//     PlcTask Inputs/GVL_iXlinker.EtherCAT_Master_BKCUCX.TcTerminals210_EK1100_1.TcTerminals210_1BK1250.A_0132_KL_1032_2_Ch_Input_48V_3_0ms.Channel_1.Input <-> Channel 1/Input
//     PlcTask Inputs/GVL_iXlinker.EtherCAT_Master_BKCUCX.TcTerminals210_EK1100_1.TcTerminals210_1BK1250.A_0132_KL_1032_2_Ch_Input_48V_3_0ms.Channel_2.Input <-> Channel 2/Input
//   PLC/PLC Instance <-> EtherCAT Master BKCUCX/TcTerminals210_EK1100_1/TcTerminals210_1BK1250/A_0133(KL 1052, 2 Ch. Input +/- (24V, 3.0ms))
//     PlcTask Inputs/GVL_iXlinker.EtherCAT_Master_BKCUCX.TcTerminals210_EK1100_1.TcTerminals210_1BK1250.A_0133_KL_1052_2_Ch_Input_24V_3_0ms.Channel_1.Input <-> Channel 1/Input
//     PlcTask Inputs/GVL_iXlinker.EtherCAT_Master_BKCUCX.TcTerminals210_EK1100_1.TcTerminals210_1BK1250.A_0133_KL_1052_2_Ch_Input_24V_3_0ms.Channel_2.Input <-> Channel 2/Input
//   PLC/PLC Instance <-> EtherCAT Master BKCUCX/TcTerminals210_EK1100_1/TcTerminals210_1BK1250/A_0134(KL 1104, 4 Ch. Input (24V, 3.0ms))
//     PlcTask Inputs/GVL_iXlinker.EtherCAT_Master_BKCUCX.TcTerminals210_EK1100_1.TcTerminals210_1BK1250.A_0134_KL_1104_4_Ch_Input_24V_3_0ms.Channel_1.Input <-> Channel 1/Input
//     PlcTask Inputs/GVL_iXlinker.EtherCAT_Master_BKCUCX.TcTerminals210_EK1100_1.TcTerminals210_1BK1250.A_0134_KL_1104_4_Ch_Input_24V_3_0ms.Channel_2.Input <-> Channel 2/Input
//     PlcTask Inputs/GVL_iXlinker.EtherCAT_Master_BKCUCX.TcTerminals210_EK1100_1.TcTerminals210_1BK1250.A_0134_KL_1104_4_Ch_Input_24V_3_0ms.Channel_3.Input <-> Channel 3/Input
//     PlcTask Inputs/GVL_iXlinker.EtherCAT_Master_BKCUCX.TcTerminals210_EK1100_1.TcTerminals210_1BK1250.A_0134_KL_1104_4_Ch_Input_24V_3_0ms.Channel_4.Input <-> Channel 4/Input
//   PLC/PLC Instance <-> EtherCAT Master BKCUCX/TcTerminals210_EK1100_1/TcTerminals210_1BK1250/A_0135(KL 1114, 4 Ch. Input (24V, 0.2ms))
//     PlcTask Inputs/GVL_iXlinker.EtherCAT_Master_BKCUCX.TcTerminals210_EK1100_1.TcTerminals210_1BK1250.A_0135_KL_1114_4_Ch_Input_24V_0_2ms.Channel_1.Input <-> Channel 1/Input
//     PlcTask Inputs/GVL_iXlinker.EtherCAT_Master_BKCUCX.TcTerminals210_EK1100_1.TcTerminals210_1BK1250.A_0135_KL_1114_4_Ch_Input_24V_0_2ms.Channel_2.Input <-> Channel 2/Input
//     PlcTask Inputs/GVL_iXlinker.EtherCAT_Master_BKCUCX.TcTerminals210_EK1100_1.TcTerminals210_1BK1250.A_0135_KL_1114_4_Ch_Input_24V_0_2ms.Channel_3.Input <-> Channel 3/Input
//     PlcTask Inputs/GVL_iXlinker.EtherCAT_Master_BKCUCX.TcTerminals210_EK1100_1.TcTerminals210_1BK1250.A_0135_KL_1114_4_Ch_Input_24V_0_2ms.Channel_4.Input <-> Channel 4/Input
//   PLC/PLC Instance <-> EtherCAT Master BKCUCX/TcTerminals210_EK1100_1/TcTerminals210_1BK1250/A_0136(KL 1124, 4 Ch. Input (5V, 0.2ms))
//     PlcTask Inputs/GVL_iXlinker.EtherCAT_Master_BKCUCX.TcTerminals210_EK1100_1.TcTerminals210_1BK1250.A_0136_KL_1124_4_Ch_Input_5V_0_2ms.Channel_1.Input <-> Channel 1/Input
//     PlcTask Inputs/GVL_iXlinker.EtherCAT_Master_BKCUCX.TcTerminals210_EK1100_1.TcTerminals210_1BK1250.A_0136_KL_1124_4_Ch_Input_5V_0_2ms.Channel_2.Input <-> Channel 2/Input
//     PlcTask Inputs/GVL_iXlinker.EtherCAT_Master_BKCUCX.TcTerminals210_EK1100_1.TcTerminals210_1BK1250.A_0136_KL_1124_4_Ch_Input_5V_0_2ms.Channel_3.Input <-> Channel 3/Input
//     PlcTask Inputs/GVL_iXlinker.EtherCAT_Master_BKCUCX.TcTerminals210_EK1100_1.TcTerminals210_1BK1250.A_0136_KL_1124_4_Ch_Input_5V_0_2ms.Channel_4.Input <-> Channel 4/Input
//   PLC/PLC Instance <-> EtherCAT Master BKCUCX/TcTerminals210_EK1100_1/TcTerminals210_1BK1250/A_0137(KL 1154, 4 Ch. Input +/- (24V, 3.0ms))
//     PlcTask Inputs/GVL_iXlinker.EtherCAT_Master_BKCUCX.TcTerminals210_EK1100_1.TcTerminals210_1BK1250.A_0137_KL_1154_4_Ch_Input_24V_3_0ms.Channel_1.Input <-> Channel 1/Input
//     PlcTask Inputs/GVL_iXlinker.EtherCAT_Master_BKCUCX.TcTerminals210_EK1100_1.TcTerminals210_1BK1250.A_0137_KL_1154_4_Ch_Input_24V_3_0ms.Channel_2.Input <-> Channel 2/Input
//     PlcTask Inputs/GVL_iXlinker.EtherCAT_Master_BKCUCX.TcTerminals210_EK1100_1.TcTerminals210_1BK1250.A_0137_KL_1154_4_Ch_Input_24V_3_0ms.Channel_3.Input <-> Channel 3/Input
//     PlcTask Inputs/GVL_iXlinker.EtherCAT_Master_BKCUCX.TcTerminals210_EK1100_1.TcTerminals210_1BK1250.A_0137_KL_1154_4_Ch_Input_24V_3_0ms.Channel_4.Input <-> Channel 4/Input
//   PLC/PLC Instance <-> EtherCAT Master BKCUCX/TcTerminals210_EK1100_1/TcTerminals210_1BK1250/A_0138(KL 1164, 4 Ch. Input +/- (24V, 0.2ms))
//     PlcTask Inputs/GVL_iXlinker.EtherCAT_Master_BKCUCX.TcTerminals210_EK1100_1.TcTerminals210_1BK1250.A_0138_KL_1164_4_Ch_Input_24V_0_2ms.Channel_1.Input <-> Channel 1/Input
//     PlcTask Inputs/GVL_iXlinker.EtherCAT_Master_BKCUCX.TcTerminals210_EK1100_1.TcTerminals210_1BK1250.A_0138_KL_1164_4_Ch_Input_24V_0_2ms.Channel_2.Input <-> Channel 2/Input
//     PlcTask Inputs/GVL_iXlinker.EtherCAT_Master_BKCUCX.TcTerminals210_EK1100_1.TcTerminals210_1BK1250.A_0138_KL_1164_4_Ch_Input_24V_0_2ms.Channel_3.Input <-> Channel 3/Input
//     PlcTask Inputs/GVL_iXlinker.EtherCAT_Master_BKCUCX.TcTerminals210_EK1100_1.TcTerminals210_1BK1250.A_0138_KL_1164_4_Ch_Input_24V_0_2ms.Channel_4.Input <-> Channel 4/Input
//   PLC/PLC Instance <-> EtherCAT Master BKCUCX/TcTerminals210_EK1100_1/TcTerminals210_1BK1250/A_0139(KL 1184, 4 Ch. Input neg. (24V, 3.0ms))
//     PlcTask Inputs/GVL_iXlinker.EtherCAT_Master_BKCUCX.TcTerminals210_EK1100_1.TcTerminals210_1BK1250.A_0139_KL_1184_4_Ch_Input_neg_24V_3_0ms.Channel_1.Input <-> Channel 1/Input
//     PlcTask Inputs/GVL_iXlinker.EtherCAT_Master_BKCUCX.TcTerminals210_EK1100_1.TcTerminals210_1BK1250.A_0139_KL_1184_4_Ch_Input_neg_24V_3_0ms.Channel_2.Input <-> Channel 2/Input
//     PlcTask Inputs/GVL_iXlinker.EtherCAT_Master_BKCUCX.TcTerminals210_EK1100_1.TcTerminals210_1BK1250.A_0139_KL_1184_4_Ch_Input_neg_24V_3_0ms.Channel_3.Input <-> Channel 3/Input
//     PlcTask Inputs/GVL_iXlinker.EtherCAT_Master_BKCUCX.TcTerminals210_EK1100_1.TcTerminals210_1BK1250.A_0139_KL_1184_4_Ch_Input_neg_24V_3_0ms.Channel_4.Input <-> Channel 4/Input
//   PLC/PLC Instance <-> EtherCAT Master BKCUCX/TcTerminals210_EK1100_1/TcTerminals210_1BK1250/A_0140(KL 1194, 4 Ch. Input neg. (24V, 0.2ms))
//     PlcTask Inputs/GVL_iXlinker.EtherCAT_Master_BKCUCX.TcTerminals210_EK1100_1.TcTerminals210_1BK1250.A_0140_KL_1194_4_Ch_Input_neg_24V_0_2ms.Channel_1.Input <-> Channel 1/Input
//     PlcTask Inputs/GVL_iXlinker.EtherCAT_Master_BKCUCX.TcTerminals210_EK1100_1.TcTerminals210_1BK1250.A_0140_KL_1194_4_Ch_Input_neg_24V_0_2ms.Channel_2.Input <-> Channel 2/Input
//     PlcTask Inputs/GVL_iXlinker.EtherCAT_Master_BKCUCX.TcTerminals210_EK1100_1.TcTerminals210_1BK1250.A_0140_KL_1194_4_Ch_Input_neg_24V_0_2ms.Channel_3.Input <-> Channel 3/Input
//     PlcTask Inputs/GVL_iXlinker.EtherCAT_Master_BKCUCX.TcTerminals210_EK1100_1.TcTerminals210_1BK1250.A_0140_KL_1194_4_Ch_Input_neg_24V_0_2ms.Channel_4.Input <-> Channel 4/Input
//   PLC/PLC Instance <-> EtherCAT Master BKCUCX/TcTerminals210_EK1100_1/TcTerminals210_1BK1250/A_0141(KL 1212, 2 Ch. Input (24V, with Power))
//     PlcTask Inputs/GVL_iXlinker.EtherCAT_Master_BKCUCX.TcTerminals210_EK1100_1.TcTerminals210_1BK1250.A_0141_KL_1212_2_Ch_Input_24V_with_Power.Channel_1.Input <-> Channel 1/Input
//     PlcTask Inputs/GVL_iXlinker.EtherCAT_Master_BKCUCX.TcTerminals210_EK1100_1.TcTerminals210_1BK1250.A_0141_KL_1212_2_Ch_Input_24V_with_Power.Channel_2.Input <-> Channel 2/Input
//     PlcTask Inputs/GVL_iXlinker.EtherCAT_Master_BKCUCX.TcTerminals210_EK1100_1.TcTerminals210_1BK1250.A_0141_KL_1212_2_Ch_Input_24V_with_Power.Channel_1.Error <-> Channel 1/Error
//     PlcTask Inputs/GVL_iXlinker.EtherCAT_Master_BKCUCX.TcTerminals210_EK1100_1.TcTerminals210_1BK1250.A_0141_KL_1212_2_Ch_Input_24V_with_Power.Channel_2.Error <-> Channel 2/Error
//     PlcTask Outputs/GVL_iXlinker.EtherCAT_Master_BKCUCX.TcTerminals210_EK1100_1.TcTerminals210_1BK1250.A_0141_KL_1212_2_Ch_Input_24V_with_Power.Channel_1.Power <-> Channel 1/Power
//     PlcTask Outputs/GVL_iXlinker.EtherCAT_Master_BKCUCX.TcTerminals210_EK1100_1.TcTerminals210_1BK1250.A_0141_KL_1212_2_Ch_Input_24V_with_Power.Channel_2.Power <-> Channel 2/Power
//   PLC/PLC Instance <-> EtherCAT Master BKCUCX/TcTerminals210_EK1100_1/TcTerminals210_1BK1250/A_0142(KL 1232, 2 Ch. Input (24V, edge triggered puls expansion))
//     PlcTask Inputs/GVL_iXlinker.EtherCAT_Master_BKCUCX.TcTerminals210_EK1100_1.TcTerminals210_1BK1250.A_0142_KL_1232_2_Ch_Input_24V_edge_triggered_puls_expansion.Channel_1.Input <-> Channel 1/Input
//     PlcTask Inputs/GVL_iXlinker.EtherCAT_Master_BKCUCX.TcTerminals210_EK1100_1.TcTerminals210_1BK1250.A_0142_KL_1232_2_Ch_Input_24V_edge_triggered_puls_expansion.Channel_2.Input <-> Channel 2/Input
//   PLC/PLC Instance <-> EtherCAT Master BKCUCX/TcTerminals210_EK1100_1/TcTerminals210_1BK1250/A_0143(KL 1302, 2 Ch. Input (24V, 3.0ms, 6mA))
//     PlcTask Inputs/GVL_iXlinker.EtherCAT_Master_BKCUCX.TcTerminals210_EK1100_1.TcTerminals210_1BK1250.A_0143_KL_1302_2_Ch_Input_24V_3_0ms_6mA.Channel_1.Input <-> Channel 1/Input
//     PlcTask Inputs/GVL_iXlinker.EtherCAT_Master_BKCUCX.TcTerminals210_EK1100_1.TcTerminals210_1BK1250.A_0143_KL_1302_2_Ch_Input_24V_3_0ms_6mA.Channel_2.Input <-> Channel 2/Input
//   PLC/PLC Instance <-> EtherCAT Master BKCUCX/TcTerminals210_EK1100_1/TcTerminals210_1BK1250/A_0144(KL 1304, 4 Ch. Input (24V, 3.0ms, 6mA))
//     PlcTask Inputs/GVL_iXlinker.EtherCAT_Master_BKCUCX.TcTerminals210_EK1100_1.TcTerminals210_1BK1250.A_0144_KL_1304_4_Ch_Input_24V_3_0ms_6mA.Channel_1.Input <-> Channel 1/Input
//     PlcTask Inputs/GVL_iXlinker.EtherCAT_Master_BKCUCX.TcTerminals210_EK1100_1.TcTerminals210_1BK1250.A_0144_KL_1304_4_Ch_Input_24V_3_0ms_6mA.Channel_2.Input <-> Channel 2/Input
//     PlcTask Inputs/GVL_iXlinker.EtherCAT_Master_BKCUCX.TcTerminals210_EK1100_1.TcTerminals210_1BK1250.A_0144_KL_1304_4_Ch_Input_24V_3_0ms_6mA.Channel_3.Input <-> Channel 3/Input
//     PlcTask Inputs/GVL_iXlinker.EtherCAT_Master_BKCUCX.TcTerminals210_EK1100_1.TcTerminals210_1BK1250.A_0144_KL_1304_4_Ch_Input_24V_3_0ms_6mA.Channel_4.Input <-> Channel 4/Input
//   PLC/PLC Instance <-> EtherCAT Master BKCUCX/TcTerminals210_EK1100_1/TcTerminals210_1BK1250/A_0145(KL 1312, 2 Ch. Input (24V, 0.2ms, 6mA))
//     PlcTask Inputs/GVL_iXlinker.EtherCAT_Master_BKCUCX.TcTerminals210_EK1100_1.TcTerminals210_1BK1250.A_0145_KL_1312_2_Ch_Input_24V_0_2ms_6mA.Channel_1.Input <-> Channel 1/Input
//     PlcTask Inputs/GVL_iXlinker.EtherCAT_Master_BKCUCX.TcTerminals210_EK1100_1.TcTerminals210_1BK1250.A_0145_KL_1312_2_Ch_Input_24V_0_2ms_6mA.Channel_2.Input <-> Channel 2/Input
//   PLC/PLC Instance <-> EtherCAT Master BKCUCX/TcTerminals210_EK1100_1/TcTerminals210_1BK1250/A_0146(KL 1314, 4 Ch. Input (24V, 0.2ms, 6mA))
//     PlcTask Inputs/GVL_iXlinker.EtherCAT_Master_BKCUCX.TcTerminals210_EK1100_1.TcTerminals210_1BK1250.A_0146_KL_1314_4_Ch_Input_24V_0_2ms_6mA.Channel_1.Input <-> Channel 1/Input
//     PlcTask Inputs/GVL_iXlinker.EtherCAT_Master_BKCUCX.TcTerminals210_EK1100_1.TcTerminals210_1BK1250.A_0146_KL_1314_4_Ch_Input_24V_0_2ms_6mA.Channel_2.Input <-> Channel 2/Input
//     PlcTask Inputs/GVL_iXlinker.EtherCAT_Master_BKCUCX.TcTerminals210_EK1100_1.TcTerminals210_1BK1250.A_0146_KL_1314_4_Ch_Input_24V_0_2ms_6mA.Channel_3.Input <-> Channel 3/Input
//     PlcTask Inputs/GVL_iXlinker.EtherCAT_Master_BKCUCX.TcTerminals210_EK1100_1.TcTerminals210_1BK1250.A_0146_KL_1314_4_Ch_Input_24V_0_2ms_6mA.Channel_4.Input <-> Channel 4/Input
//   PLC/PLC Instance <-> EtherCAT Master BKCUCX/TcTerminals210_EK1100_1/TcTerminals210_1BK1250/A_0147(KL 1352, 2 Ch. Input (24V, 3.0ms, NAMUR))
//     PlcTask Inputs/GVL_iXlinker.EtherCAT_Master_BKCUCX.TcTerminals210_EK1100_1.TcTerminals210_1BK1250.A_0147_KL_1352_2_Ch_Input_24V_3_0ms_NAMUR.Channel_1.Input <-> Channel 1/Input
//     PlcTask Inputs/GVL_iXlinker.EtherCAT_Master_BKCUCX.TcTerminals210_EK1100_1.TcTerminals210_1BK1250.A_0147_KL_1352_2_Ch_Input_24V_3_0ms_NAMUR.Channel_2.Input <-> Channel 2/Input
//     PlcTask Inputs/GVL_iXlinker.EtherCAT_Master_BKCUCX.TcTerminals210_EK1100_1.TcTerminals210_1BK1250.A_0147_KL_1352_2_Ch_Input_24V_3_0ms_NAMUR.Channel_1.Error <-> Channel 1/Error
//     PlcTask Inputs/GVL_iXlinker.EtherCAT_Master_BKCUCX.TcTerminals210_EK1100_1.TcTerminals210_1BK1250.A_0147_KL_1352_2_Ch_Input_24V_3_0ms_NAMUR.Channel_2.Error <-> Channel 2/Error
//   PLC/PLC Instance <-> EtherCAT Master BKCUCX/TcTerminals210_EK1100_1/TcTerminals210_1BK1250/A_0148(KL 1362, 2 Ch. Input (24V, for break-in alarm))
//     PlcTask Inputs/GVL_iXlinker.EtherCAT_Master_BKCUCX.TcTerminals210_EK1100_1.TcTerminals210_1BK1250.A_0148_KL_1362_2_Ch_Input_24V_for_break_in_alarm.Channel_1.Input <-> Channel 1/Input
//     PlcTask Inputs/GVL_iXlinker.EtherCAT_Master_BKCUCX.TcTerminals210_EK1100_1.TcTerminals210_1BK1250.A_0148_KL_1362_2_Ch_Input_24V_for_break_in_alarm.Channel_2.Input <-> Channel 2/Input
//     PlcTask Inputs/GVL_iXlinker.EtherCAT_Master_BKCUCX.TcTerminals210_EK1100_1.TcTerminals210_1BK1250.A_0148_KL_1362_2_Ch_Input_24V_for_break_in_alarm.Channel_1.Error <-> Channel 1/Error
//     PlcTask Inputs/GVL_iXlinker.EtherCAT_Master_BKCUCX.TcTerminals210_EK1100_1.TcTerminals210_1BK1250.A_0148_KL_1362_2_Ch_Input_24V_for_break_in_alarm.Channel_2.Error <-> Channel 2/Error
//   PLC/PLC Instance <-> EtherCAT Master BKCUCX/TcTerminals210_EK1100_1/TcTerminals210_1BK1250/A_0149(KL 1382, 2 Ch. Input (24V, thermistor sensors))
//     PlcTask Inputs/GVL_iXlinker.EtherCAT_Master_BKCUCX.TcTerminals210_EK1100_1.TcTerminals210_1BK1250.A_0149_KL_1382_2_Ch_Input_24V_thermistor_sensors.Channel_1.Input <-> Channel 1/Input
//     PlcTask Inputs/GVL_iXlinker.EtherCAT_Master_BKCUCX.TcTerminals210_EK1100_1.TcTerminals210_1BK1250.A_0149_KL_1382_2_Ch_Input_24V_thermistor_sensors.Channel_2.Input <-> Channel 2/Input
//     PlcTask Inputs/GVL_iXlinker.EtherCAT_Master_BKCUCX.TcTerminals210_EK1100_1.TcTerminals210_1BK1250.A_0149_KL_1382_2_Ch_Input_24V_thermistor_sensors.Channel_1.Error <-> Channel 1/Error
//     PlcTask Inputs/GVL_iXlinker.EtherCAT_Master_BKCUCX.TcTerminals210_EK1100_1.TcTerminals210_1BK1250.A_0149_KL_1382_2_Ch_Input_24V_thermistor_sensors.Channel_2.Error <-> Channel 2/Error
//   PLC/PLC Instance <-> EtherCAT Master BKCUCX/TcTerminals210_EK1100_1/TcTerminals210_1BK1250/A_0150(KL 1402, 2 Ch. Input (24V, 3.0ms, type 3))
//     PlcTask Inputs/GVL_iXlinker.EtherCAT_Master_BKCUCX.TcTerminals210_EK1100_1.TcTerminals210_1BK1250.A_0150_KL_1402_2_Ch_Input_24V_3_0ms_type_3.Channel_1.Input <-> Channel 1/Input
//     PlcTask Inputs/GVL_iXlinker.EtherCAT_Master_BKCUCX.TcTerminals210_EK1100_1.TcTerminals210_1BK1250.A_0150_KL_1402_2_Ch_Input_24V_3_0ms_type_3.Channel_2.Input <-> Channel 2/Input
//   PLC/PLC Instance <-> EtherCAT Master BKCUCX/TcTerminals210_EK1100_1/TcTerminals210_1BK1250/A_0151(KL 1404, 4 Ch. Input (24V, 3.0ms, 3mA, 2 wire))
//     PlcTask Inputs/GVL_iXlinker.EtherCAT_Master_BKCUCX.TcTerminals210_EK1100_1.TcTerminals210_1BK1250.A_0151_KL_1404_4_Ch_Input_24V_3_0ms_3mA_2_wire.Channel_1.Input <-> Channel 1/Input
//     PlcTask Inputs/GVL_iXlinker.EtherCAT_Master_BKCUCX.TcTerminals210_EK1100_1.TcTerminals210_1BK1250.A_0151_KL_1404_4_Ch_Input_24V_3_0ms_3mA_2_wire.Channel_2.Input <-> Channel 2/Input
//     PlcTask Inputs/GVL_iXlinker.EtherCAT_Master_BKCUCX.TcTerminals210_EK1100_1.TcTerminals210_1BK1250.A_0151_KL_1404_4_Ch_Input_24V_3_0ms_3mA_2_wire.Channel_3.Input <-> Channel 3/Input
//     PlcTask Inputs/GVL_iXlinker.EtherCAT_Master_BKCUCX.TcTerminals210_EK1100_1.TcTerminals210_1BK1250.A_0151_KL_1404_4_Ch_Input_24V_3_0ms_3mA_2_wire.Channel_4.Input <-> Channel 4/Input
//   PLC/PLC Instance <-> EtherCAT Master BKCUCX/TcTerminals210_EK1100_1/TcTerminals210_1BK1250/A_0152(KL 1408, 8 Ch. Input (24V, 3.0ms))
//     PlcTask Inputs/GVL_iXlinker.EtherCAT_Master_BKCUCX.TcTerminals210_EK1100_1.TcTerminals210_1BK1250.A_0152_KL_1408_8_Ch_Input_24V_3_0ms.Channel_1.Input <-> Channel 1/Input
//     PlcTask Inputs/GVL_iXlinker.EtherCAT_Master_BKCUCX.TcTerminals210_EK1100_1.TcTerminals210_1BK1250.A_0152_KL_1408_8_Ch_Input_24V_3_0ms.Channel_2.Input <-> Channel 2/Input
//     PlcTask Inputs/GVL_iXlinker.EtherCAT_Master_BKCUCX.TcTerminals210_EK1100_1.TcTerminals210_1BK1250.A_0152_KL_1408_8_Ch_Input_24V_3_0ms.Channel_3.Input <-> Channel 3/Input
//     PlcTask Inputs/GVL_iXlinker.EtherCAT_Master_BKCUCX.TcTerminals210_EK1100_1.TcTerminals210_1BK1250.A_0152_KL_1408_8_Ch_Input_24V_3_0ms.Channel_4.Input <-> Channel 4/Input
//     PlcTask Inputs/GVL_iXlinker.EtherCAT_Master_BKCUCX.TcTerminals210_EK1100_1.TcTerminals210_1BK1250.A_0152_KL_1408_8_Ch_Input_24V_3_0ms.Channel_5.Input <-> Channel 5/Input
//     PlcTask Inputs/GVL_iXlinker.EtherCAT_Master_BKCUCX.TcTerminals210_EK1100_1.TcTerminals210_1BK1250.A_0152_KL_1408_8_Ch_Input_24V_3_0ms.Channel_6.Input <-> Channel 6/Input
//     PlcTask Inputs/GVL_iXlinker.EtherCAT_Master_BKCUCX.TcTerminals210_EK1100_1.TcTerminals210_1BK1250.A_0152_KL_1408_8_Ch_Input_24V_3_0ms.Channel_7.Input <-> Channel 7/Input
//     PlcTask Inputs/GVL_iXlinker.EtherCAT_Master_BKCUCX.TcTerminals210_EK1100_1.TcTerminals210_1BK1250.A_0152_KL_1408_8_Ch_Input_24V_3_0ms.Channel_8.Input <-> Channel 8/Input
//   PLC/PLC Instance <-> EtherCAT Master BKCUCX/TcTerminals210_EK1100_1/TcTerminals210_1BK1250/A_0153(KL 1412, 2 Ch. Input (24V, 0.2ms, type 3))
//     PlcTask Inputs/GVL_iXlinker.EtherCAT_Master_BKCUCX.TcTerminals210_EK1100_1.TcTerminals210_1BK1250.A_0153_KL_1412_2_Ch_Input_24V_0_2ms_type_3.Channel_1.Input <-> Channel 1/Input
//     PlcTask Inputs/GVL_iXlinker.EtherCAT_Master_BKCUCX.TcTerminals210_EK1100_1.TcTerminals210_1BK1250.A_0153_KL_1412_2_Ch_Input_24V_0_2ms_type_3.Channel_2.Input <-> Channel 2/Input
//   PLC/PLC Instance <-> EtherCAT Master BKCUCX/TcTerminals210_EK1100_1/TcTerminals210_1BK1250/A_0154(KL 1414, 4 Ch. Input (24V, 0.2ms, 3mA, 2 wire))
//     PlcTask Inputs/GVL_iXlinker.EtherCAT_Master_BKCUCX.TcTerminals210_EK1100_1.TcTerminals210_1BK1250.A_0154_KL_1414_4_Ch_Input_24V_0_2ms_3mA_2_wire.Channel_1.Input <-> Channel 1/Input
//     PlcTask Inputs/GVL_iXlinker.EtherCAT_Master_BKCUCX.TcTerminals210_EK1100_1.TcTerminals210_1BK1250.A_0154_KL_1414_4_Ch_Input_24V_0_2ms_3mA_2_wire.Channel_2.Input <-> Channel 2/Input
//     PlcTask Inputs/GVL_iXlinker.EtherCAT_Master_BKCUCX.TcTerminals210_EK1100_1.TcTerminals210_1BK1250.A_0154_KL_1414_4_Ch_Input_24V_0_2ms_3mA_2_wire.Channel_3.Input <-> Channel 3/Input
//     PlcTask Inputs/GVL_iXlinker.EtherCAT_Master_BKCUCX.TcTerminals210_EK1100_1.TcTerminals210_1BK1250.A_0154_KL_1414_4_Ch_Input_24V_0_2ms_3mA_2_wire.Channel_4.Input <-> Channel 4/Input
//   PLC/PLC Instance <-> EtherCAT Master BKCUCX/TcTerminals210_EK1100_1/TcTerminals210_1BK1250/A_0155(KL 1418, 8 Ch. Input (24V, 0.2ms))
//     PlcTask Inputs/GVL_iXlinker.EtherCAT_Master_BKCUCX.TcTerminals210_EK1100_1.TcTerminals210_1BK1250.A_0155_KL_1418_8_Ch_Input_24V_0_2ms.Channel_1.Input <-> Channel 1/Input
//     PlcTask Inputs/GVL_iXlinker.EtherCAT_Master_BKCUCX.TcTerminals210_EK1100_1.TcTerminals210_1BK1250.A_0155_KL_1418_8_Ch_Input_24V_0_2ms.Channel_2.Input <-> Channel 2/Input
//     PlcTask Inputs/GVL_iXlinker.EtherCAT_Master_BKCUCX.TcTerminals210_EK1100_1.TcTerminals210_1BK1250.A_0155_KL_1418_8_Ch_Input_24V_0_2ms.Channel_3.Input <-> Channel 3/Input
//     PlcTask Inputs/GVL_iXlinker.EtherCAT_Master_BKCUCX.TcTerminals210_EK1100_1.TcTerminals210_1BK1250.A_0155_KL_1418_8_Ch_Input_24V_0_2ms.Channel_4.Input <-> Channel 4/Input
//     PlcTask Inputs/GVL_iXlinker.EtherCAT_Master_BKCUCX.TcTerminals210_EK1100_1.TcTerminals210_1BK1250.A_0155_KL_1418_8_Ch_Input_24V_0_2ms.Channel_5.Input <-> Channel 5/Input
//     PlcTask Inputs/GVL_iXlinker.EtherCAT_Master_BKCUCX.TcTerminals210_EK1100_1.TcTerminals210_1BK1250.A_0155_KL_1418_8_Ch_Input_24V_0_2ms.Channel_6.Input <-> Channel 6/Input
//     PlcTask Inputs/GVL_iXlinker.EtherCAT_Master_BKCUCX.TcTerminals210_EK1100_1.TcTerminals210_1BK1250.A_0155_KL_1418_8_Ch_Input_24V_0_2ms.Channel_7.Input <-> Channel 7/Input
//     PlcTask Inputs/GVL_iXlinker.EtherCAT_Master_BKCUCX.TcTerminals210_EK1100_1.TcTerminals210_1BK1250.A_0155_KL_1418_8_Ch_Input_24V_0_2ms.Channel_8.Input <-> Channel 8/Input
//   PLC/PLC Instance <-> EtherCAT Master BKCUCX/TcTerminals210_EK1100_1/TcTerminals210_1BK1250/A_0156(KL 1434, 4 Ch. Input (24V, 0.2ms, 6mA, 2 wire))
//     PlcTask Inputs/GVL_iXlinker.EtherCAT_Master_BKCUCX.TcTerminals210_EK1100_1.TcTerminals210_1BK1250.A_0156_KL_1434_4_Ch_Input_24V_0_2ms_6mA_2_wire.Channel_1.Input <-> Channel 1/Input
//     PlcTask Inputs/GVL_iXlinker.EtherCAT_Master_BKCUCX.TcTerminals210_EK1100_1.TcTerminals210_1BK1250.A_0156_KL_1434_4_Ch_Input_24V_0_2ms_6mA_2_wire.Channel_2.Input <-> Channel 2/Input
//     PlcTask Inputs/GVL_iXlinker.EtherCAT_Master_BKCUCX.TcTerminals210_EK1100_1.TcTerminals210_1BK1250.A_0156_KL_1434_4_Ch_Input_24V_0_2ms_6mA_2_wire.Channel_3.Input <-> Channel 3/Input
//     PlcTask Inputs/GVL_iXlinker.EtherCAT_Master_BKCUCX.TcTerminals210_EK1100_1.TcTerminals210_1BK1250.A_0156_KL_1434_4_Ch_Input_24V_0_2ms_6mA_2_wire.Channel_4.Input <-> Channel 4/Input
//   PLC/PLC Instance <-> EtherCAT Master BKCUCX/TcTerminals210_EK1100_1/TcTerminals210_1BK1250/A_0157(KL 1488, 8 Ch. Input (24V neg, 3ms))
//     PlcTask Inputs/GVL_iXlinker.EtherCAT_Master_BKCUCX.TcTerminals210_EK1100_1.TcTerminals210_1BK1250.A_0157_KL_1488_8_Ch_Input_24V_neg_3ms.Channel_1.Input <-> Channel 1/Input
//     PlcTask Inputs/GVL_iXlinker.EtherCAT_Master_BKCUCX.TcTerminals210_EK1100_1.TcTerminals210_1BK1250.A_0157_KL_1488_8_Ch_Input_24V_neg_3ms.Channel_2.Input <-> Channel 2/Input
//     PlcTask Inputs/GVL_iXlinker.EtherCAT_Master_BKCUCX.TcTerminals210_EK1100_1.TcTerminals210_1BK1250.A_0157_KL_1488_8_Ch_Input_24V_neg_3ms.Channel_3.Input <-> Channel 3/Input
//     PlcTask Inputs/GVL_iXlinker.EtherCAT_Master_BKCUCX.TcTerminals210_EK1100_1.TcTerminals210_1BK1250.A_0157_KL_1488_8_Ch_Input_24V_neg_3ms.Channel_4.Input <-> Channel 4/Input
//     PlcTask Inputs/GVL_iXlinker.EtherCAT_Master_BKCUCX.TcTerminals210_EK1100_1.TcTerminals210_1BK1250.A_0157_KL_1488_8_Ch_Input_24V_neg_3ms.Channel_5.Input <-> Channel 5/Input
//     PlcTask Inputs/GVL_iXlinker.EtherCAT_Master_BKCUCX.TcTerminals210_EK1100_1.TcTerminals210_1BK1250.A_0157_KL_1488_8_Ch_Input_24V_neg_3ms.Channel_6.Input <-> Channel 6/Input
//     PlcTask Inputs/GVL_iXlinker.EtherCAT_Master_BKCUCX.TcTerminals210_EK1100_1.TcTerminals210_1BK1250.A_0157_KL_1488_8_Ch_Input_24V_neg_3ms.Channel_7.Input <-> Channel 7/Input
//     PlcTask Inputs/GVL_iXlinker.EtherCAT_Master_BKCUCX.TcTerminals210_EK1100_1.TcTerminals210_1BK1250.A_0157_KL_1488_8_Ch_Input_24V_neg_3ms.Channel_8.Input <-> Channel 8/Input
//   PLC/PLC Instance <-> EtherCAT Master BKCUCX/TcTerminals210_EK1100_1/TcTerminals210_1BK1250/A_0158(KL 1498, 8 Ch. Input (24V neg, 0.2ms))
//     PlcTask Inputs/GVL_iXlinker.EtherCAT_Master_BKCUCX.TcTerminals210_EK1100_1.TcTerminals210_1BK1250.A_0158_KL_1498_8_Ch_Input_24V_neg_0_2ms.Channel_1.Input <-> Channel 1/Input
//     PlcTask Inputs/GVL_iXlinker.EtherCAT_Master_BKCUCX.TcTerminals210_EK1100_1.TcTerminals210_1BK1250.A_0158_KL_1498_8_Ch_Input_24V_neg_0_2ms.Channel_2.Input <-> Channel 2/Input
//     PlcTask Inputs/GVL_iXlinker.EtherCAT_Master_BKCUCX.TcTerminals210_EK1100_1.TcTerminals210_1BK1250.A_0158_KL_1498_8_Ch_Input_24V_neg_0_2ms.Channel_3.Input <-> Channel 3/Input
//     PlcTask Inputs/GVL_iXlinker.EtherCAT_Master_BKCUCX.TcTerminals210_EK1100_1.TcTerminals210_1BK1250.A_0158_KL_1498_8_Ch_Input_24V_neg_0_2ms.Channel_4.Input <-> Channel 4/Input
//     PlcTask Inputs/GVL_iXlinker.EtherCAT_Master_BKCUCX.TcTerminals210_EK1100_1.TcTerminals210_1BK1250.A_0158_KL_1498_8_Ch_Input_24V_neg_0_2ms.Channel_5.Input <-> Channel 5/Input
//     PlcTask Inputs/GVL_iXlinker.EtherCAT_Master_BKCUCX.TcTerminals210_EK1100_1.TcTerminals210_1BK1250.A_0158_KL_1498_8_Ch_Input_24V_neg_0_2ms.Channel_6.Input <-> Channel 6/Input
//     PlcTask Inputs/GVL_iXlinker.EtherCAT_Master_BKCUCX.TcTerminals210_EK1100_1.TcTerminals210_1BK1250.A_0158_KL_1498_8_Ch_Input_24V_neg_0_2ms.Channel_7.Input <-> Channel 7/Input
//     PlcTask Inputs/GVL_iXlinker.EtherCAT_Master_BKCUCX.TcTerminals210_EK1100_1.TcTerminals210_1BK1250.A_0158_KL_1498_8_Ch_Input_24V_neg_0_2ms.Channel_8.Input <-> Channel 8/Input
//   PLC/PLC Instance <-> EtherCAT Master BKCUCX/TcTerminals210_EK1100_1/TcTerminals210_1BK1250/A_0159(KL 1501, 1 Ch. +/- Counter)
//     PlcTask Inputs/GVL_iXlinker.EtherCAT_Master_BKCUCX.TcTerminals210_EK1100_1.TcTerminals210_1BK1250.A_0159_KL_1501_1_Ch_Counter.Channel_1.State <-> Channel 1/State
//     PlcTask Inputs/GVL_iXlinker.EtherCAT_Master_BKCUCX.TcTerminals210_EK1100_1.TcTerminals210_1BK1250.A_0159_KL_1501_1_Ch_Counter.Channel_1.Data_In <-> Channel 1/Data In
//     PlcTask Outputs/GVL_iXlinker.EtherCAT_Master_BKCUCX.TcTerminals210_EK1100_1.TcTerminals210_1BK1250.A_0159_KL_1501_1_Ch_Counter.Channel_1.Ctrl <-> Channel 1/Ctrl
//     PlcTask Outputs/GVL_iXlinker.EtherCAT_Master_BKCUCX.TcTerminals210_EK1100_1.TcTerminals210_1BK1250.A_0159_KL_1501_1_Ch_Counter.Channel_1.Data_Out <-> Channel 1/Data Out
//   PLC/PLC Instance <-> EtherCAT Master BKCUCX/TcTerminals210_EK1100_1/TcTerminals210_1BK1250/A_0161(KL 1501-1002)
//     PlcTask Inputs/GVL_iXlinker.EtherCAT_Master_BKCUCX.TcTerminals210_EK1100_1.TcTerminals210_1BK1250.A_0161_KL_1501_1002.Channel_1.Status <-> Channel 1/Status
//     PlcTask Inputs/GVL_iXlinker.EtherCAT_Master_BKCUCX.TcTerminals210_EK1100_1.TcTerminals210_1BK1250.A_0161_KL_1501_1002.Channel_1.Counter <-> Channel 1/Counter
//     PlcTask Inputs/GVL_iXlinker.EtherCAT_Master_BKCUCX.TcTerminals210_EK1100_1.TcTerminals210_1BK1250.A_0161_KL_1501_1002.Channel_1.Latch_PeriodL <-> Channel 1/Latch/PeriodL
//     PlcTask Inputs/GVL_iXlinker.EtherCAT_Master_BKCUCX.TcTerminals210_EK1100_1.TcTerminals210_1BK1250.A_0161_KL_1501_1002.Channel_1.PeriodH <-> Channel 1/PeriodH
//     PlcTask Outputs/GVL_iXlinker.EtherCAT_Master_BKCUCX.TcTerminals210_EK1100_1.TcTerminals210_1BK1250.A_0161_KL_1501_1002.Channel_1.Ctrl <-> Channel 1/Ctrl
//     PlcTask Outputs/GVL_iXlinker.EtherCAT_Master_BKCUCX.TcTerminals210_EK1100_1.TcTerminals210_1BK1250.A_0161_KL_1501_1002.Channel_1.RegData <-> Channel 1/RegData
//   PLC/PLC Instance <-> EtherCAT Master BKCUCX/TcTerminals210_EK1100_1/TcTerminals210_1BK1250/A_0162(KL 1512, 2 Ch. +/- Counter)
//     PlcTask Inputs/GVL_iXlinker.EtherCAT_Master_BKCUCX.TcTerminals210_EK1100_1.TcTerminals210_1BK1250.A_0162_KL_1512_2_Ch_Counter.Channel_1.State <-> Channel 1/State
//     PlcTask Inputs/GVL_iXlinker.EtherCAT_Master_BKCUCX.TcTerminals210_EK1100_1.TcTerminals210_1BK1250.A_0162_KL_1512_2_Ch_Counter.Channel_2.State <-> Channel 2/State
//     PlcTask Inputs/GVL_iXlinker.EtherCAT_Master_BKCUCX.TcTerminals210_EK1100_1.TcTerminals210_1BK1250.A_0162_KL_1512_2_Ch_Counter.Channel_1.Data_In <-> Channel 1/Data In
//     PlcTask Inputs/GVL_iXlinker.EtherCAT_Master_BKCUCX.TcTerminals210_EK1100_1.TcTerminals210_1BK1250.A_0162_KL_1512_2_Ch_Counter.Channel_2.Data_In <-> Channel 2/Data In
//     PlcTask Outputs/GVL_iXlinker.EtherCAT_Master_BKCUCX.TcTerminals210_EK1100_1.TcTerminals210_1BK1250.A_0162_KL_1512_2_Ch_Counter.Channel_1.Ctrl <-> Channel 1/Ctrl
//     PlcTask Outputs/GVL_iXlinker.EtherCAT_Master_BKCUCX.TcTerminals210_EK1100_1.TcTerminals210_1BK1250.A_0162_KL_1512_2_Ch_Counter.Channel_2.Ctrl <-> Channel 2/Ctrl
//     PlcTask Outputs/GVL_iXlinker.EtherCAT_Master_BKCUCX.TcTerminals210_EK1100_1.TcTerminals210_1BK1250.A_0162_KL_1512_2_Ch_Counter.Channel_1.Data_Out <-> Channel 1/Data Out
//     PlcTask Outputs/GVL_iXlinker.EtherCAT_Master_BKCUCX.TcTerminals210_EK1100_1.TcTerminals210_1BK1250.A_0162_KL_1512_2_Ch_Counter.Channel_2.Data_Out <-> Channel 2/Data Out
//   PLC/PLC Instance <-> EtherCAT Master BKCUCX/TcTerminals210_EK1100_1/TcTerminals210_1BK1250/A_0163(KL 1702, 2 Ch. Input (230V, 10.0ms))
//     PlcTask Inputs/GVL_iXlinker.EtherCAT_Master_BKCUCX.TcTerminals210_EK1100_1.TcTerminals210_1BK1250.A_0163_KL_1702_2_Ch_Input_230V_10_0ms.Channel_1.Input <-> Channel 1/Input
//     PlcTask Inputs/GVL_iXlinker.EtherCAT_Master_BKCUCX.TcTerminals210_EK1100_1.TcTerminals210_1BK1250.A_0163_KL_1702_2_Ch_Input_230V_10_0ms.Channel_2.Input <-> Channel 2/Input
//   PLC/PLC Instance <-> EtherCAT Master BKCUCX/TcTerminals210_EK1100_1/TcTerminals210_1BK1250/A_0164(KL 1704, 4 Ch. Input (230V, 10.0ms))
//     PlcTask Inputs/GVL_iXlinker.EtherCAT_Master_BKCUCX.TcTerminals210_EK1100_1.TcTerminals210_1BK1250.A_0164_KL_1704_4_Ch_Input_230V_10_0ms.Channel_1.Input <-> Channel 1/Input
//     PlcTask Inputs/GVL_iXlinker.EtherCAT_Master_BKCUCX.TcTerminals210_EK1100_1.TcTerminals210_1BK1250.A_0164_KL_1704_4_Ch_Input_230V_10_0ms.Channel_2.Input <-> Channel 2/Input
//     PlcTask Inputs/GVL_iXlinker.EtherCAT_Master_BKCUCX.TcTerminals210_EK1100_1.TcTerminals210_1BK1250.A_0164_KL_1704_4_Ch_Input_230V_10_0ms.Channel_3.Input <-> Channel 3/Input
//     PlcTask Inputs/GVL_iXlinker.EtherCAT_Master_BKCUCX.TcTerminals210_EK1100_1.TcTerminals210_1BK1250.A_0164_KL_1704_4_Ch_Input_230V_10_0ms.Channel_4.Input <-> Channel 4/Input
//   PLC/PLC Instance <-> EtherCAT Master BKCUCX/TcTerminals210_EK1100_1/TcTerminals210_1BK1250/A_0165(KL 1712, 2 Ch. Input (120V, 10.0ms))
//     PlcTask Inputs/GVL_iXlinker.EtherCAT_Master_BKCUCX.TcTerminals210_EK1100_1.TcTerminals210_1BK1250.A_0165_KL_1712_2_Ch_Input_120V_10_0ms.Channel_1.Input <-> Channel 1/Input
//     PlcTask Inputs/GVL_iXlinker.EtherCAT_Master_BKCUCX.TcTerminals210_EK1100_1.TcTerminals210_1BK1250.A_0165_KL_1712_2_Ch_Input_120V_10_0ms.Channel_2.Input <-> Channel 2/Input
//   PLC/PLC Instance <-> EtherCAT Master BKCUCX/TcTerminals210_EK1100_1/TcTerminals210_1BK1250/A_0166(KL 1712-0060, 2 Ch. Input (60V, 10.0ms))
//     PlcTask Inputs/GVL_iXlinker.EtherCAT_Master_BKCUCX.TcTerminals210_EK1100_1.TcTerminals210_1BK1250.A_0166_KL_1712_0060_2_Ch_Input_60V_10_0ms.Channel_1.Input <-> Channel 1/Input
//     PlcTask Inputs/GVL_iXlinker.EtherCAT_Master_BKCUCX.TcTerminals210_EK1100_1.TcTerminals210_1BK1250.A_0166_KL_1712_0060_2_Ch_Input_60V_10_0ms.Channel_2.Input <-> Channel 2/Input
//   PLC/PLC Instance <-> EtherCAT Master BKCUCX/TcTerminals210_EK1100_1/TcTerminals210_1BK1250/A_0167(KL 1722, 2 Ch. Input (230V, 10.0ms, no power contacts))
//     PlcTask Inputs/GVL_iXlinker.EtherCAT_Master_BKCUCX.TcTerminals210_EK1100_1.TcTerminals210_1BK1250.A_0167_KL_1722_2_Ch_Input_230V_10_0ms_no_power_contacts.Channel_1.Input <-> Channel 1/Input
//     PlcTask Inputs/GVL_iXlinker.EtherCAT_Master_BKCUCX.TcTerminals210_EK1100_1.TcTerminals210_1BK1250.A_0167_KL_1722_2_Ch_Input_230V_10_0ms_no_power_contacts.Channel_2.Input <-> Channel 2/Input
//   PLC/PLC Instance <-> EtherCAT Master BKCUCX/TcTerminals210_EK1100_1/TcTerminals210_1BK1250/A_0168(KL 1804, 4 Ch. Input (24V, 3.0ms, 3 wire))
//     PlcTask Inputs/GVL_iXlinker.EtherCAT_Master_BKCUCX.TcTerminals210_EK1100_1.TcTerminals210_1BK1250.A_0168_KL_1804_4_Ch_Input_24V_3_0ms_3_wire.Channel_1.Input <-> Channel 1/Input
//     PlcTask Inputs/GVL_iXlinker.EtherCAT_Master_BKCUCX.TcTerminals210_EK1100_1.TcTerminals210_1BK1250.A_0168_KL_1804_4_Ch_Input_24V_3_0ms_3_wire.Channel_2.Input <-> Channel 2/Input
//     PlcTask Inputs/GVL_iXlinker.EtherCAT_Master_BKCUCX.TcTerminals210_EK1100_1.TcTerminals210_1BK1250.A_0168_KL_1804_4_Ch_Input_24V_3_0ms_3_wire.Channel_3.Input <-> Channel 3/Input
//     PlcTask Inputs/GVL_iXlinker.EtherCAT_Master_BKCUCX.TcTerminals210_EK1100_1.TcTerminals210_1BK1250.A_0168_KL_1804_4_Ch_Input_24V_3_0ms_3_wire.Channel_4.Input <-> Channel 4/Input
//   PLC/PLC Instance <-> EtherCAT Master BKCUCX/TcTerminals210_EK1100_1/TcTerminals210_1BK1250/A_0169(KL 1808, 8 Ch. Input (24V, 3.0ms, 2 wire))
//     PlcTask Inputs/GVL_iXlinker.EtherCAT_Master_BKCUCX.TcTerminals210_EK1100_1.TcTerminals210_1BK1250.A_0169_KL_1808_8_Ch_Input_24V_3_0ms_2_wire.Channel_1.Input <-> Channel 1/Input
//     PlcTask Inputs/GVL_iXlinker.EtherCAT_Master_BKCUCX.TcTerminals210_EK1100_1.TcTerminals210_1BK1250.A_0169_KL_1808_8_Ch_Input_24V_3_0ms_2_wire.Channel_2.Input <-> Channel 2/Input
//     PlcTask Inputs/GVL_iXlinker.EtherCAT_Master_BKCUCX.TcTerminals210_EK1100_1.TcTerminals210_1BK1250.A_0169_KL_1808_8_Ch_Input_24V_3_0ms_2_wire.Channel_3.Input <-> Channel 3/Input
//     PlcTask Inputs/GVL_iXlinker.EtherCAT_Master_BKCUCX.TcTerminals210_EK1100_1.TcTerminals210_1BK1250.A_0169_KL_1808_8_Ch_Input_24V_3_0ms_2_wire.Channel_4.Input <-> Channel 4/Input
//     PlcTask Inputs/GVL_iXlinker.EtherCAT_Master_BKCUCX.TcTerminals210_EK1100_1.TcTerminals210_1BK1250.A_0169_KL_1808_8_Ch_Input_24V_3_0ms_2_wire.Channel_5.Input <-> Channel 5/Input
//     PlcTask Inputs/GVL_iXlinker.EtherCAT_Master_BKCUCX.TcTerminals210_EK1100_1.TcTerminals210_1BK1250.A_0169_KL_1808_8_Ch_Input_24V_3_0ms_2_wire.Channel_6.Input <-> Channel 6/Input
//     PlcTask Inputs/GVL_iXlinker.EtherCAT_Master_BKCUCX.TcTerminals210_EK1100_1.TcTerminals210_1BK1250.A_0169_KL_1808_8_Ch_Input_24V_3_0ms_2_wire.Channel_7.Input <-> Channel 7/Input
//     PlcTask Inputs/GVL_iXlinker.EtherCAT_Master_BKCUCX.TcTerminals210_EK1100_1.TcTerminals210_1BK1250.A_0169_KL_1808_8_Ch_Input_24V_3_0ms_2_wire.Channel_8.Input <-> Channel 8/Input
//   PLC/PLC Instance <-> EtherCAT Master BKCUCX/TcTerminals210_EK1100_1/TcTerminals210_1BK1250/A_0170(KL 1809, 16 Ch. Input (24V, 3.0ms))
//     PlcTask Inputs/GVL_iXlinker.EtherCAT_Master_BKCUCX.TcTerminals210_EK1100_1.TcTerminals210_1BK1250.A_0170_KL_1809_16_Ch_Input_24V_3_0ms.Channel_1.Input <-> Channel 1/Input
//     PlcTask Inputs/GVL_iXlinker.EtherCAT_Master_BKCUCX.TcTerminals210_EK1100_1.TcTerminals210_1BK1250.A_0170_KL_1809_16_Ch_Input_24V_3_0ms.Channel_2.Input <-> Channel 2/Input
//     PlcTask Inputs/GVL_iXlinker.EtherCAT_Master_BKCUCX.TcTerminals210_EK1100_1.TcTerminals210_1BK1250.A_0170_KL_1809_16_Ch_Input_24V_3_0ms.Channel_3.Input <-> Channel 3/Input
//     PlcTask Inputs/GVL_iXlinker.EtherCAT_Master_BKCUCX.TcTerminals210_EK1100_1.TcTerminals210_1BK1250.A_0170_KL_1809_16_Ch_Input_24V_3_0ms.Channel_4.Input <-> Channel 4/Input
//     PlcTask Inputs/GVL_iXlinker.EtherCAT_Master_BKCUCX.TcTerminals210_EK1100_1.TcTerminals210_1BK1250.A_0170_KL_1809_16_Ch_Input_24V_3_0ms.Channel_5.Input <-> Channel 5/Input
//     PlcTask Inputs/GVL_iXlinker.EtherCAT_Master_BKCUCX.TcTerminals210_EK1100_1.TcTerminals210_1BK1250.A_0170_KL_1809_16_Ch_Input_24V_3_0ms.Channel_6.Input <-> Channel 6/Input
//     PlcTask Inputs/GVL_iXlinker.EtherCAT_Master_BKCUCX.TcTerminals210_EK1100_1.TcTerminals210_1BK1250.A_0170_KL_1809_16_Ch_Input_24V_3_0ms.Channel_7.Input <-> Channel 7/Input
//     PlcTask Inputs/GVL_iXlinker.EtherCAT_Master_BKCUCX.TcTerminals210_EK1100_1.TcTerminals210_1BK1250.A_0170_KL_1809_16_Ch_Input_24V_3_0ms.Channel_8.Input <-> Channel 8/Input
//     PlcTask Inputs/GVL_iXlinker.EtherCAT_Master_BKCUCX.TcTerminals210_EK1100_1.TcTerminals210_1BK1250.A_0170_KL_1809_16_Ch_Input_24V_3_0ms.Channel_9.Input <-> Channel 9/Input
//     PlcTask Inputs/GVL_iXlinker.EtherCAT_Master_BKCUCX.TcTerminals210_EK1100_1.TcTerminals210_1BK1250.A_0170_KL_1809_16_Ch_Input_24V_3_0ms.Channel_10.Input <-> Channel 10/Input
//     PlcTask Inputs/GVL_iXlinker.EtherCAT_Master_BKCUCX.TcTerminals210_EK1100_1.TcTerminals210_1BK1250.A_0170_KL_1809_16_Ch_Input_24V_3_0ms.Channel_11.Input <-> Channel 11/Input
//     PlcTask Inputs/GVL_iXlinker.EtherCAT_Master_BKCUCX.TcTerminals210_EK1100_1.TcTerminals210_1BK1250.A_0170_KL_1809_16_Ch_Input_24V_3_0ms.Channel_12.Input <-> Channel 12/Input
//     PlcTask Inputs/GVL_iXlinker.EtherCAT_Master_BKCUCX.TcTerminals210_EK1100_1.TcTerminals210_1BK1250.A_0170_KL_1809_16_Ch_Input_24V_3_0ms.Channel_13.Input <-> Channel 13/Input
//     PlcTask Inputs/GVL_iXlinker.EtherCAT_Master_BKCUCX.TcTerminals210_EK1100_1.TcTerminals210_1BK1250.A_0170_KL_1809_16_Ch_Input_24V_3_0ms.Channel_14.Input <-> Channel 14/Input
//     PlcTask Inputs/GVL_iXlinker.EtherCAT_Master_BKCUCX.TcTerminals210_EK1100_1.TcTerminals210_1BK1250.A_0170_KL_1809_16_Ch_Input_24V_3_0ms.Channel_15.Input <-> Channel 15/Input
//     PlcTask Inputs/GVL_iXlinker.EtherCAT_Master_BKCUCX.TcTerminals210_EK1100_1.TcTerminals210_1BK1250.A_0170_KL_1809_16_Ch_Input_24V_3_0ms.Channel_16.Input <-> Channel 16/Input
//   PLC/PLC Instance <-> EtherCAT Master BKCUCX/TcTerminals210_EK1100_1/TcTerminals210_1BK1250/A_0171(KL 1814, 4 Ch. Input (24V, 0.2ms, 3 wire))
//     PlcTask Inputs/GVL_iXlinker.EtherCAT_Master_BKCUCX.TcTerminals210_EK1100_1.TcTerminals210_1BK1250.A_0171_KL_1814_4_Ch_Input_24V_0_2ms_3_wire.Channel_1.Input <-> Channel 1/Input
//     PlcTask Inputs/GVL_iXlinker.EtherCAT_Master_BKCUCX.TcTerminals210_EK1100_1.TcTerminals210_1BK1250.A_0171_KL_1814_4_Ch_Input_24V_0_2ms_3_wire.Channel_2.Input <-> Channel 2/Input
//     PlcTask Inputs/GVL_iXlinker.EtherCAT_Master_BKCUCX.TcTerminals210_EK1100_1.TcTerminals210_1BK1250.A_0171_KL_1814_4_Ch_Input_24V_0_2ms_3_wire.Channel_3.Input <-> Channel 3/Input
//     PlcTask Inputs/GVL_iXlinker.EtherCAT_Master_BKCUCX.TcTerminals210_EK1100_1.TcTerminals210_1BK1250.A_0171_KL_1814_4_Ch_Input_24V_0_2ms_3_wire.Channel_4.Input <-> Channel 4/Input
//   PLC/PLC Instance <-> EtherCAT Master BKCUCX/TcTerminals210_EK1100_1/TcTerminals210_1BK1250/A_0172(KL 1819, 16 Ch. Input (24V, 0.2ms))
//     PlcTask Inputs/GVL_iXlinker.EtherCAT_Master_BKCUCX.TcTerminals210_EK1100_1.TcTerminals210_1BK1250.A_0172_KL_1819_16_Ch_Input_24V_0_2ms.Channel_1.Input <-> Channel 1/Input
//     PlcTask Inputs/GVL_iXlinker.EtherCAT_Master_BKCUCX.TcTerminals210_EK1100_1.TcTerminals210_1BK1250.A_0172_KL_1819_16_Ch_Input_24V_0_2ms.Channel_2.Input <-> Channel 2/Input
//     PlcTask Inputs/GVL_iXlinker.EtherCAT_Master_BKCUCX.TcTerminals210_EK1100_1.TcTerminals210_1BK1250.A_0172_KL_1819_16_Ch_Input_24V_0_2ms.Channel_3.Input <-> Channel 3/Input
//     PlcTask Inputs/GVL_iXlinker.EtherCAT_Master_BKCUCX.TcTerminals210_EK1100_1.TcTerminals210_1BK1250.A_0172_KL_1819_16_Ch_Input_24V_0_2ms.Channel_4.Input <-> Channel 4/Input
//     PlcTask Inputs/GVL_iXlinker.EtherCAT_Master_BKCUCX.TcTerminals210_EK1100_1.TcTerminals210_1BK1250.A_0172_KL_1819_16_Ch_Input_24V_0_2ms.Channel_5.Input <-> Channel 5/Input
//     PlcTask Inputs/GVL_iXlinker.EtherCAT_Master_BKCUCX.TcTerminals210_EK1100_1.TcTerminals210_1BK1250.A_0172_KL_1819_16_Ch_Input_24V_0_2ms.Channel_6.Input <-> Channel 6/Input
//     PlcTask Inputs/GVL_iXlinker.EtherCAT_Master_BKCUCX.TcTerminals210_EK1100_1.TcTerminals210_1BK1250.A_0172_KL_1819_16_Ch_Input_24V_0_2ms.Channel_7.Input <-> Channel 7/Input
//     PlcTask Inputs/GVL_iXlinker.EtherCAT_Master_BKCUCX.TcTerminals210_EK1100_1.TcTerminals210_1BK1250.A_0172_KL_1819_16_Ch_Input_24V_0_2ms.Channel_8.Input <-> Channel 8/Input
//     PlcTask Inputs/GVL_iXlinker.EtherCAT_Master_BKCUCX.TcTerminals210_EK1100_1.TcTerminals210_1BK1250.A_0172_KL_1819_16_Ch_Input_24V_0_2ms.Channel_9.Input <-> Channel 9/Input
//     PlcTask Inputs/GVL_iXlinker.EtherCAT_Master_BKCUCX.TcTerminals210_EK1100_1.TcTerminals210_1BK1250.A_0172_KL_1819_16_Ch_Input_24V_0_2ms.Channel_10.Input <-> Channel 10/Input
//     PlcTask Inputs/GVL_iXlinker.EtherCAT_Master_BKCUCX.TcTerminals210_EK1100_1.TcTerminals210_1BK1250.A_0172_KL_1819_16_Ch_Input_24V_0_2ms.Channel_11.Input <-> Channel 11/Input
//     PlcTask Inputs/GVL_iXlinker.EtherCAT_Master_BKCUCX.TcTerminals210_EK1100_1.TcTerminals210_1BK1250.A_0172_KL_1819_16_Ch_Input_24V_0_2ms.Channel_12.Input <-> Channel 12/Input
//     PlcTask Inputs/GVL_iXlinker.EtherCAT_Master_BKCUCX.TcTerminals210_EK1100_1.TcTerminals210_1BK1250.A_0172_KL_1819_16_Ch_Input_24V_0_2ms.Channel_13.Input <-> Channel 13/Input
//     PlcTask Inputs/GVL_iXlinker.EtherCAT_Master_BKCUCX.TcTerminals210_EK1100_1.TcTerminals210_1BK1250.A_0172_KL_1819_16_Ch_Input_24V_0_2ms.Channel_14.Input <-> Channel 14/Input
//     PlcTask Inputs/GVL_iXlinker.EtherCAT_Master_BKCUCX.TcTerminals210_EK1100_1.TcTerminals210_1BK1250.A_0172_KL_1819_16_Ch_Input_24V_0_2ms.Channel_15.Input <-> Channel 15/Input
//     PlcTask Inputs/GVL_iXlinker.EtherCAT_Master_BKCUCX.TcTerminals210_EK1100_1.TcTerminals210_1BK1250.A_0172_KL_1819_16_Ch_Input_24V_0_2ms.Channel_16.Input <-> Channel 16/Input
//   PLC/PLC Instance <-> EtherCAT Master BKCUCX/TcTerminals210_EK1100_1/TcTerminals210_1BK1250/A_0173(KL 1859, 8 Ch. In-/Output (24V, 3.0ms, 0.5A))
//     PlcTask Inputs/GVL_iXlinker.EtherCAT_Master_BKCUCX.TcTerminals210_EK1100_1.TcTerminals210_1BK1250.A_0173_KL_1859_8_Ch_In_Output_24V_3_0ms_0_5A.Channel_1.Input <-> Channel 1/Input
//     PlcTask Inputs/GVL_iXlinker.EtherCAT_Master_BKCUCX.TcTerminals210_EK1100_1.TcTerminals210_1BK1250.A_0173_KL_1859_8_Ch_In_Output_24V_3_0ms_0_5A.Channel_2.Input <-> Channel 2/Input
//     PlcTask Inputs/GVL_iXlinker.EtherCAT_Master_BKCUCX.TcTerminals210_EK1100_1.TcTerminals210_1BK1250.A_0173_KL_1859_8_Ch_In_Output_24V_3_0ms_0_5A.Channel_3.Input <-> Channel 3/Input
//     PlcTask Inputs/GVL_iXlinker.EtherCAT_Master_BKCUCX.TcTerminals210_EK1100_1.TcTerminals210_1BK1250.A_0173_KL_1859_8_Ch_In_Output_24V_3_0ms_0_5A.Channel_4.Input <-> Channel 4/Input
//     PlcTask Inputs/GVL_iXlinker.EtherCAT_Master_BKCUCX.TcTerminals210_EK1100_1.TcTerminals210_1BK1250.A_0173_KL_1859_8_Ch_In_Output_24V_3_0ms_0_5A.Channel_5.Input <-> Channel 5/Input
//     PlcTask Inputs/GVL_iXlinker.EtherCAT_Master_BKCUCX.TcTerminals210_EK1100_1.TcTerminals210_1BK1250.A_0173_KL_1859_8_Ch_In_Output_24V_3_0ms_0_5A.Channel_6.Input <-> Channel 6/Input
//     PlcTask Inputs/GVL_iXlinker.EtherCAT_Master_BKCUCX.TcTerminals210_EK1100_1.TcTerminals210_1BK1250.A_0173_KL_1859_8_Ch_In_Output_24V_3_0ms_0_5A.Channel_7.Input <-> Channel 7/Input
//     PlcTask Inputs/GVL_iXlinker.EtherCAT_Master_BKCUCX.TcTerminals210_EK1100_1.TcTerminals210_1BK1250.A_0173_KL_1859_8_Ch_In_Output_24V_3_0ms_0_5A.Channel_8.Input <-> Channel 8/Input
//     PlcTask Outputs/GVL_iXlinker.EtherCAT_Master_BKCUCX.TcTerminals210_EK1100_1.TcTerminals210_1BK1250.A_0173_KL_1859_8_Ch_In_Output_24V_3_0ms_0_5A.Channel_1.Output <-> Channel 1/Output
//     PlcTask Outputs/GVL_iXlinker.EtherCAT_Master_BKCUCX.TcTerminals210_EK1100_1.TcTerminals210_1BK1250.A_0173_KL_1859_8_Ch_In_Output_24V_3_0ms_0_5A.Channel_2.Output <-> Channel 2/Output
//     PlcTask Outputs/GVL_iXlinker.EtherCAT_Master_BKCUCX.TcTerminals210_EK1100_1.TcTerminals210_1BK1250.A_0173_KL_1859_8_Ch_In_Output_24V_3_0ms_0_5A.Channel_3.Output <-> Channel 3/Output
//     PlcTask Outputs/GVL_iXlinker.EtherCAT_Master_BKCUCX.TcTerminals210_EK1100_1.TcTerminals210_1BK1250.A_0173_KL_1859_8_Ch_In_Output_24V_3_0ms_0_5A.Channel_4.Output <-> Channel 4/Output
//     PlcTask Outputs/GVL_iXlinker.EtherCAT_Master_BKCUCX.TcTerminals210_EK1100_1.TcTerminals210_1BK1250.A_0173_KL_1859_8_Ch_In_Output_24V_3_0ms_0_5A.Channel_5.Output <-> Channel 5/Output
//     PlcTask Outputs/GVL_iXlinker.EtherCAT_Master_BKCUCX.TcTerminals210_EK1100_1.TcTerminals210_1BK1250.A_0173_KL_1859_8_Ch_In_Output_24V_3_0ms_0_5A.Channel_6.Output <-> Channel 6/Output
//     PlcTask Outputs/GVL_iXlinker.EtherCAT_Master_BKCUCX.TcTerminals210_EK1100_1.TcTerminals210_1BK1250.A_0173_KL_1859_8_Ch_In_Output_24V_3_0ms_0_5A.Channel_7.Output <-> Channel 7/Output
//     PlcTask Outputs/GVL_iXlinker.EtherCAT_Master_BKCUCX.TcTerminals210_EK1100_1.TcTerminals210_1BK1250.A_0173_KL_1859_8_Ch_In_Output_24V_3_0ms_0_5A.Channel_8.Output <-> Channel 8/Output
//   PLC/PLC Instance <-> EtherCAT Master BKCUCX/TcTerminals210_EK1100_1/TcTerminals210_1BK1250/A_0174(KL 1862, 16 Ch. Input (24V, 3.0ms, flat ribbon))
//     PlcTask Inputs/GVL_iXlinker.EtherCAT_Master_BKCUCX.TcTerminals210_EK1100_1.TcTerminals210_1BK1250.A_0174_KL_1862_16_Ch_Input_24V_3_0ms_flat_ribbon.Channel_1.Input <-> Channel 1/Input
//     PlcTask Inputs/GVL_iXlinker.EtherCAT_Master_BKCUCX.TcTerminals210_EK1100_1.TcTerminals210_1BK1250.A_0174_KL_1862_16_Ch_Input_24V_3_0ms_flat_ribbon.Channel_2.Input <-> Channel 2/Input
//     PlcTask Inputs/GVL_iXlinker.EtherCAT_Master_BKCUCX.TcTerminals210_EK1100_1.TcTerminals210_1BK1250.A_0174_KL_1862_16_Ch_Input_24V_3_0ms_flat_ribbon.Channel_3.Input <-> Channel 3/Input
//     PlcTask Inputs/GVL_iXlinker.EtherCAT_Master_BKCUCX.TcTerminals210_EK1100_1.TcTerminals210_1BK1250.A_0174_KL_1862_16_Ch_Input_24V_3_0ms_flat_ribbon.Channel_4.Input <-> Channel 4/Input
//     PlcTask Inputs/GVL_iXlinker.EtherCAT_Master_BKCUCX.TcTerminals210_EK1100_1.TcTerminals210_1BK1250.A_0174_KL_1862_16_Ch_Input_24V_3_0ms_flat_ribbon.Channel_5.Input <-> Channel 5/Input
//     PlcTask Inputs/GVL_iXlinker.EtherCAT_Master_BKCUCX.TcTerminals210_EK1100_1.TcTerminals210_1BK1250.A_0174_KL_1862_16_Ch_Input_24V_3_0ms_flat_ribbon.Channel_6.Input <-> Channel 6/Input
//     PlcTask Inputs/GVL_iXlinker.EtherCAT_Master_BKCUCX.TcTerminals210_EK1100_1.TcTerminals210_1BK1250.A_0174_KL_1862_16_Ch_Input_24V_3_0ms_flat_ribbon.Channel_7.Input <-> Channel 7/Input
//     PlcTask Inputs/GVL_iXlinker.EtherCAT_Master_BKCUCX.TcTerminals210_EK1100_1.TcTerminals210_1BK1250.A_0174_KL_1862_16_Ch_Input_24V_3_0ms_flat_ribbon.Channel_8.Input <-> Channel 8/Input
//     PlcTask Inputs/GVL_iXlinker.EtherCAT_Master_BKCUCX.TcTerminals210_EK1100_1.TcTerminals210_1BK1250.A_0174_KL_1862_16_Ch_Input_24V_3_0ms_flat_ribbon.Channel_9.Input <-> Channel 9/Input
//     PlcTask Inputs/GVL_iXlinker.EtherCAT_Master_BKCUCX.TcTerminals210_EK1100_1.TcTerminals210_1BK1250.A_0174_KL_1862_16_Ch_Input_24V_3_0ms_flat_ribbon.Channel_10.Input <-> Channel 10/Input
//     PlcTask Inputs/GVL_iXlinker.EtherCAT_Master_BKCUCX.TcTerminals210_EK1100_1.TcTerminals210_1BK1250.A_0174_KL_1862_16_Ch_Input_24V_3_0ms_flat_ribbon.Channel_11.Input <-> Channel 11/Input
//     PlcTask Inputs/GVL_iXlinker.EtherCAT_Master_BKCUCX.TcTerminals210_EK1100_1.TcTerminals210_1BK1250.A_0174_KL_1862_16_Ch_Input_24V_3_0ms_flat_ribbon.Channel_12.Input <-> Channel 12/Input
//     PlcTask Inputs/GVL_iXlinker.EtherCAT_Master_BKCUCX.TcTerminals210_EK1100_1.TcTerminals210_1BK1250.A_0174_KL_1862_16_Ch_Input_24V_3_0ms_flat_ribbon.Channel_13.Input <-> Channel 13/Input
//     PlcTask Inputs/GVL_iXlinker.EtherCAT_Master_BKCUCX.TcTerminals210_EK1100_1.TcTerminals210_1BK1250.A_0174_KL_1862_16_Ch_Input_24V_3_0ms_flat_ribbon.Channel_14.Input <-> Channel 14/Input
//     PlcTask Inputs/GVL_iXlinker.EtherCAT_Master_BKCUCX.TcTerminals210_EK1100_1.TcTerminals210_1BK1250.A_0174_KL_1862_16_Ch_Input_24V_3_0ms_flat_ribbon.Channel_15.Input <-> Channel 15/Input
//     PlcTask Inputs/GVL_iXlinker.EtherCAT_Master_BKCUCX.TcTerminals210_EK1100_1.TcTerminals210_1BK1250.A_0174_KL_1862_16_Ch_Input_24V_3_0ms_flat_ribbon.Channel_16.Input <-> Channel 16/Input
//   PLC/PLC Instance <-> EtherCAT Master BKCUCX/TcTerminals210_EK1100_1/TcTerminals210_1BK1250/A_0175(KL 1862-0010, 16 Ch. Input (24V, 3.0ms, flat ribbon, ground switching))
//     PlcTask Inputs/GVL_iXlinker.EtherCAT_Master_BKCUCX.TcTerminals210_EK1100_1.TcTerminals210_1BK1250.A_0175_KL_1862_0010_16_Ch_Input_24V_3_0ms_flat_ribbon_ground_switching.Channel_1.Input <-> Channel 1/Input
//     PlcTask Inputs/GVL_iXlinker.EtherCAT_Master_BKCUCX.TcTerminals210_EK1100_1.TcTerminals210_1BK1250.A_0175_KL_1862_0010_16_Ch_Input_24V_3_0ms_flat_ribbon_ground_switching.Channel_2.Input <-> Channel 2/Input
//     PlcTask Inputs/GVL_iXlinker.EtherCAT_Master_BKCUCX.TcTerminals210_EK1100_1.TcTerminals210_1BK1250.A_0175_KL_1862_0010_16_Ch_Input_24V_3_0ms_flat_ribbon_ground_switching.Channel_3.Input <-> Channel 3/Input
//     PlcTask Inputs/GVL_iXlinker.EtherCAT_Master_BKCUCX.TcTerminals210_EK1100_1.TcTerminals210_1BK1250.A_0175_KL_1862_0010_16_Ch_Input_24V_3_0ms_flat_ribbon_ground_switching.Channel_4.Input <-> Channel 4/Input
//     PlcTask Inputs/GVL_iXlinker.EtherCAT_Master_BKCUCX.TcTerminals210_EK1100_1.TcTerminals210_1BK1250.A_0175_KL_1862_0010_16_Ch_Input_24V_3_0ms_flat_ribbon_ground_switching.Channel_5.Input <-> Channel 5/Input
//     PlcTask Inputs/GVL_iXlinker.EtherCAT_Master_BKCUCX.TcTerminals210_EK1100_1.TcTerminals210_1BK1250.A_0175_KL_1862_0010_16_Ch_Input_24V_3_0ms_flat_ribbon_ground_switching.Channel_6.Input <-> Channel 6/Input
//     PlcTask Inputs/GVL_iXlinker.EtherCAT_Master_BKCUCX.TcTerminals210_EK1100_1.TcTerminals210_1BK1250.A_0175_KL_1862_0010_16_Ch_Input_24V_3_0ms_flat_ribbon_ground_switching.Channel_7.Input <-> Channel 7/Input
//     PlcTask Inputs/GVL_iXlinker.EtherCAT_Master_BKCUCX.TcTerminals210_EK1100_1.TcTerminals210_1BK1250.A_0175_KL_1862_0010_16_Ch_Input_24V_3_0ms_flat_ribbon_ground_switching.Channel_8.Input <-> Channel 8/Input
//     PlcTask Inputs/GVL_iXlinker.EtherCAT_Master_BKCUCX.TcTerminals210_EK1100_1.TcTerminals210_1BK1250.A_0175_KL_1862_0010_16_Ch_Input_24V_3_0ms_flat_ribbon_ground_switching.Channel_9.Input <-> Channel 9/Input
//     PlcTask Inputs/GVL_iXlinker.EtherCAT_Master_BKCUCX.TcTerminals210_EK1100_1.TcTerminals210_1BK1250.A_0175_KL_1862_0010_16_Ch_Input_24V_3_0ms_flat_ribbon_ground_switching.Channel_10.Input <-> Channel 10/Input
//     PlcTask Inputs/GVL_iXlinker.EtherCAT_Master_BKCUCX.TcTerminals210_EK1100_1.TcTerminals210_1BK1250.A_0175_KL_1862_0010_16_Ch_Input_24V_3_0ms_flat_ribbon_ground_switching.Channel_11.Input <-> Channel 11/Input
//     PlcTask Inputs/GVL_iXlinker.EtherCAT_Master_BKCUCX.TcTerminals210_EK1100_1.TcTerminals210_1BK1250.A_0175_KL_1862_0010_16_Ch_Input_24V_3_0ms_flat_ribbon_ground_switching.Channel_12.Input <-> Channel 12/Input
//     PlcTask Inputs/GVL_iXlinker.EtherCAT_Master_BKCUCX.TcTerminals210_EK1100_1.TcTerminals210_1BK1250.A_0175_KL_1862_0010_16_Ch_Input_24V_3_0ms_flat_ribbon_ground_switching.Channel_13.Input <-> Channel 13/Input
//     PlcTask Inputs/GVL_iXlinker.EtherCAT_Master_BKCUCX.TcTerminals210_EK1100_1.TcTerminals210_1BK1250.A_0175_KL_1862_0010_16_Ch_Input_24V_3_0ms_flat_ribbon_ground_switching.Channel_14.Input <-> Channel 14/Input
//     PlcTask Inputs/GVL_iXlinker.EtherCAT_Master_BKCUCX.TcTerminals210_EK1100_1.TcTerminals210_1BK1250.A_0175_KL_1862_0010_16_Ch_Input_24V_3_0ms_flat_ribbon_ground_switching.Channel_15.Input <-> Channel 15/Input
//     PlcTask Inputs/GVL_iXlinker.EtherCAT_Master_BKCUCX.TcTerminals210_EK1100_1.TcTerminals210_1BK1250.A_0175_KL_1862_0010_16_Ch_Input_24V_3_0ms_flat_ribbon_ground_switching.Channel_16.Input <-> Channel 16/Input
//   PLC/PLC Instance <-> EtherCAT Master BKCUCX/TcTerminals210_EK1100_1/TcTerminals210_1BK1250/A_0176(KL 1872, 16 Ch. Input (24V, 0.2ms, flat ribbon))
//     PlcTask Inputs/GVL_iXlinker.EtherCAT_Master_BKCUCX.TcTerminals210_EK1100_1.TcTerminals210_1BK1250.A_0176_KL_1872_16_Ch_Input_24V_0_2ms_flat_ribbon.Channel_1.Input <-> Channel 1/Input
//     PlcTask Inputs/GVL_iXlinker.EtherCAT_Master_BKCUCX.TcTerminals210_EK1100_1.TcTerminals210_1BK1250.A_0176_KL_1872_16_Ch_Input_24V_0_2ms_flat_ribbon.Channel_2.Input <-> Channel 2/Input
//     PlcTask Inputs/GVL_iXlinker.EtherCAT_Master_BKCUCX.TcTerminals210_EK1100_1.TcTerminals210_1BK1250.A_0176_KL_1872_16_Ch_Input_24V_0_2ms_flat_ribbon.Channel_3.Input <-> Channel 3/Input
//     PlcTask Inputs/GVL_iXlinker.EtherCAT_Master_BKCUCX.TcTerminals210_EK1100_1.TcTerminals210_1BK1250.A_0176_KL_1872_16_Ch_Input_24V_0_2ms_flat_ribbon.Channel_4.Input <-> Channel 4/Input
//     PlcTask Inputs/GVL_iXlinker.EtherCAT_Master_BKCUCX.TcTerminals210_EK1100_1.TcTerminals210_1BK1250.A_0176_KL_1872_16_Ch_Input_24V_0_2ms_flat_ribbon.Channel_5.Input <-> Channel 5/Input
//     PlcTask Inputs/GVL_iXlinker.EtherCAT_Master_BKCUCX.TcTerminals210_EK1100_1.TcTerminals210_1BK1250.A_0176_KL_1872_16_Ch_Input_24V_0_2ms_flat_ribbon.Channel_6.Input <-> Channel 6/Input
//     PlcTask Inputs/GVL_iXlinker.EtherCAT_Master_BKCUCX.TcTerminals210_EK1100_1.TcTerminals210_1BK1250.A_0176_KL_1872_16_Ch_Input_24V_0_2ms_flat_ribbon.Channel_7.Input <-> Channel 7/Input
//     PlcTask Inputs/GVL_iXlinker.EtherCAT_Master_BKCUCX.TcTerminals210_EK1100_1.TcTerminals210_1BK1250.A_0176_KL_1872_16_Ch_Input_24V_0_2ms_flat_ribbon.Channel_8.Input <-> Channel 8/Input
//     PlcTask Inputs/GVL_iXlinker.EtherCAT_Master_BKCUCX.TcTerminals210_EK1100_1.TcTerminals210_1BK1250.A_0176_KL_1872_16_Ch_Input_24V_0_2ms_flat_ribbon.Channel_9.Input <-> Channel 9/Input
//     PlcTask Inputs/GVL_iXlinker.EtherCAT_Master_BKCUCX.TcTerminals210_EK1100_1.TcTerminals210_1BK1250.A_0176_KL_1872_16_Ch_Input_24V_0_2ms_flat_ribbon.Channel_10.Input <-> Channel 10/Input
//     PlcTask Inputs/GVL_iXlinker.EtherCAT_Master_BKCUCX.TcTerminals210_EK1100_1.TcTerminals210_1BK1250.A_0176_KL_1872_16_Ch_Input_24V_0_2ms_flat_ribbon.Channel_11.Input <-> Channel 11/Input
//     PlcTask Inputs/GVL_iXlinker.EtherCAT_Master_BKCUCX.TcTerminals210_EK1100_1.TcTerminals210_1BK1250.A_0176_KL_1872_16_Ch_Input_24V_0_2ms_flat_ribbon.Channel_12.Input <-> Channel 12/Input
//     PlcTask Inputs/GVL_iXlinker.EtherCAT_Master_BKCUCX.TcTerminals210_EK1100_1.TcTerminals210_1BK1250.A_0176_KL_1872_16_Ch_Input_24V_0_2ms_flat_ribbon.Channel_13.Input <-> Channel 13/Input
//     PlcTask Inputs/GVL_iXlinker.EtherCAT_Master_BKCUCX.TcTerminals210_EK1100_1.TcTerminals210_1BK1250.A_0176_KL_1872_16_Ch_Input_24V_0_2ms_flat_ribbon.Channel_14.Input <-> Channel 14/Input
//     PlcTask Inputs/GVL_iXlinker.EtherCAT_Master_BKCUCX.TcTerminals210_EK1100_1.TcTerminals210_1BK1250.A_0176_KL_1872_16_Ch_Input_24V_0_2ms_flat_ribbon.Channel_15.Input <-> Channel 15/Input
//     PlcTask Inputs/GVL_iXlinker.EtherCAT_Master_BKCUCX.TcTerminals210_EK1100_1.TcTerminals210_1BK1250.A_0176_KL_1872_16_Ch_Input_24V_0_2ms_flat_ribbon.Channel_16.Input <-> Channel 16/Input
//   PLC/PLC Instance <-> EtherCAT Master BKCUCX/TcTerminals210_EK1100_1/TcTerminals210_1BK1250/A_0177(KL 1889, 16 Ch. Input (24V ground switching, 3.0ms))
//     PlcTask Inputs/GVL_iXlinker.EtherCAT_Master_BKCUCX.TcTerminals210_EK1100_1.TcTerminals210_1BK1250.A_0177_KL_1889_16_Ch_Input_24V_ground_switching_3_0ms.Channel_1.Input <-> Channel 1/Input
//     PlcTask Inputs/GVL_iXlinker.EtherCAT_Master_BKCUCX.TcTerminals210_EK1100_1.TcTerminals210_1BK1250.A_0177_KL_1889_16_Ch_Input_24V_ground_switching_3_0ms.Channel_2.Input <-> Channel 2/Input
//     PlcTask Inputs/GVL_iXlinker.EtherCAT_Master_BKCUCX.TcTerminals210_EK1100_1.TcTerminals210_1BK1250.A_0177_KL_1889_16_Ch_Input_24V_ground_switching_3_0ms.Channel_3.Input <-> Channel 3/Input
//     PlcTask Inputs/GVL_iXlinker.EtherCAT_Master_BKCUCX.TcTerminals210_EK1100_1.TcTerminals210_1BK1250.A_0177_KL_1889_16_Ch_Input_24V_ground_switching_3_0ms.Channel_4.Input <-> Channel 4/Input
//     PlcTask Inputs/GVL_iXlinker.EtherCAT_Master_BKCUCX.TcTerminals210_EK1100_1.TcTerminals210_1BK1250.A_0177_KL_1889_16_Ch_Input_24V_ground_switching_3_0ms.Channel_5.Input <-> Channel 5/Input
//     PlcTask Inputs/GVL_iXlinker.EtherCAT_Master_BKCUCX.TcTerminals210_EK1100_1.TcTerminals210_1BK1250.A_0177_KL_1889_16_Ch_Input_24V_ground_switching_3_0ms.Channel_6.Input <-> Channel 6/Input
//     PlcTask Inputs/GVL_iXlinker.EtherCAT_Master_BKCUCX.TcTerminals210_EK1100_1.TcTerminals210_1BK1250.A_0177_KL_1889_16_Ch_Input_24V_ground_switching_3_0ms.Channel_7.Input <-> Channel 7/Input
//     PlcTask Inputs/GVL_iXlinker.EtherCAT_Master_BKCUCX.TcTerminals210_EK1100_1.TcTerminals210_1BK1250.A_0177_KL_1889_16_Ch_Input_24V_ground_switching_3_0ms.Channel_8.Input <-> Channel 8/Input
//     PlcTask Inputs/GVL_iXlinker.EtherCAT_Master_BKCUCX.TcTerminals210_EK1100_1.TcTerminals210_1BK1250.A_0177_KL_1889_16_Ch_Input_24V_ground_switching_3_0ms.Channel_9.Input <-> Channel 9/Input
//     PlcTask Inputs/GVL_iXlinker.EtherCAT_Master_BKCUCX.TcTerminals210_EK1100_1.TcTerminals210_1BK1250.A_0177_KL_1889_16_Ch_Input_24V_ground_switching_3_0ms.Channel_10.Input <-> Channel 10/Input
//     PlcTask Inputs/GVL_iXlinker.EtherCAT_Master_BKCUCX.TcTerminals210_EK1100_1.TcTerminals210_1BK1250.A_0177_KL_1889_16_Ch_Input_24V_ground_switching_3_0ms.Channel_11.Input <-> Channel 11/Input
//     PlcTask Inputs/GVL_iXlinker.EtherCAT_Master_BKCUCX.TcTerminals210_EK1100_1.TcTerminals210_1BK1250.A_0177_KL_1889_16_Ch_Input_24V_ground_switching_3_0ms.Channel_12.Input <-> Channel 12/Input
//     PlcTask Inputs/GVL_iXlinker.EtherCAT_Master_BKCUCX.TcTerminals210_EK1100_1.TcTerminals210_1BK1250.A_0177_KL_1889_16_Ch_Input_24V_ground_switching_3_0ms.Channel_13.Input <-> Channel 13/Input
//     PlcTask Inputs/GVL_iXlinker.EtherCAT_Master_BKCUCX.TcTerminals210_EK1100_1.TcTerminals210_1BK1250.A_0177_KL_1889_16_Ch_Input_24V_ground_switching_3_0ms.Channel_14.Input <-> Channel 14/Input
//     PlcTask Inputs/GVL_iXlinker.EtherCAT_Master_BKCUCX.TcTerminals210_EK1100_1.TcTerminals210_1BK1250.A_0177_KL_1889_16_Ch_Input_24V_ground_switching_3_0ms.Channel_15.Input <-> Channel 15/Input
//     PlcTask Inputs/GVL_iXlinker.EtherCAT_Master_BKCUCX.TcTerminals210_EK1100_1.TcTerminals210_1BK1250.A_0177_KL_1889_16_Ch_Input_24V_ground_switching_3_0ms.Channel_16.Input <-> Channel 16/Input
//   PLC/PLC Instance <-> EtherCAT Master BKCUCX/TcTerminals210_EK1100_1/TcTerminals210_1BK1250/A_0178(KL 1904, 4 Ch. Safety Input)
//     PlcTask Inputs/GVL_iXlinker.EtherCAT_Master_BKCUCX.TcTerminals210_EK1100_1.TcTerminals210_1BK1250.A_0178_KL_1904_4_Ch_Safety_Input.Channel_1.Safety_In <-> Channel 1/Safety In
//     PlcTask Outputs/GVL_iXlinker.EtherCAT_Master_BKCUCX.TcTerminals210_EK1100_1.TcTerminals210_1BK1250.A_0178_KL_1904_4_Ch_Safety_Input.Channel_1.Safety_Out <-> Channel 1/Safety Out
//   PLC/PLC Instance <-> EtherCAT Master BKCUCX/TcTerminals210_EK1100_1/TcTerminals210_1BK1250/A_0179(KL 1908, 8 Ch. Safety Input)
//     PlcTask Inputs/GVL_iXlinker.EtherCAT_Master_BKCUCX.TcTerminals210_EK1100_1.TcTerminals210_1BK1250.A_0179_KL_1908_8_Ch_Safety_Input.Channel_1.Safety_In <-> Channel 1/Safety In
//     PlcTask Outputs/GVL_iXlinker.EtherCAT_Master_BKCUCX.TcTerminals210_EK1100_1.TcTerminals210_1BK1250.A_0179_KL_1908_8_Ch_Safety_Input.Channel_1.Safety_Out <-> Channel 1/Safety Out
//   PLC/PLC Instance <-> EtherCAT Master BKCUCX/TcTerminals210_EK1100_1/TcTerminals210_1BK1250/A_0180(KM 1002, 16 Ch. Input (24V, 3.0ms))
//     PlcTask Inputs/GVL_iXlinker.EtherCAT_Master_BKCUCX.TcTerminals210_EK1100_1.TcTerminals210_1BK1250.A_0180_KM_1002_16_Ch_Input_24V_3_0ms.Channel_1.Input <-> Channel 1/Input
//     PlcTask Inputs/GVL_iXlinker.EtherCAT_Master_BKCUCX.TcTerminals210_EK1100_1.TcTerminals210_1BK1250.A_0180_KM_1002_16_Ch_Input_24V_3_0ms.Channel_2.Input <-> Channel 2/Input
//     PlcTask Inputs/GVL_iXlinker.EtherCAT_Master_BKCUCX.TcTerminals210_EK1100_1.TcTerminals210_1BK1250.A_0180_KM_1002_16_Ch_Input_24V_3_0ms.Channel_3.Input <-> Channel 3/Input
//     PlcTask Inputs/GVL_iXlinker.EtherCAT_Master_BKCUCX.TcTerminals210_EK1100_1.TcTerminals210_1BK1250.A_0180_KM_1002_16_Ch_Input_24V_3_0ms.Channel_4.Input <-> Channel 4/Input
//     PlcTask Inputs/GVL_iXlinker.EtherCAT_Master_BKCUCX.TcTerminals210_EK1100_1.TcTerminals210_1BK1250.A_0180_KM_1002_16_Ch_Input_24V_3_0ms.Channel_5.Input <-> Channel 5/Input
//     PlcTask Inputs/GVL_iXlinker.EtherCAT_Master_BKCUCX.TcTerminals210_EK1100_1.TcTerminals210_1BK1250.A_0180_KM_1002_16_Ch_Input_24V_3_0ms.Channel_6.Input <-> Channel 6/Input
//     PlcTask Inputs/GVL_iXlinker.EtherCAT_Master_BKCUCX.TcTerminals210_EK1100_1.TcTerminals210_1BK1250.A_0180_KM_1002_16_Ch_Input_24V_3_0ms.Channel_7.Input <-> Channel 7/Input
//     PlcTask Inputs/GVL_iXlinker.EtherCAT_Master_BKCUCX.TcTerminals210_EK1100_1.TcTerminals210_1BK1250.A_0180_KM_1002_16_Ch_Input_24V_3_0ms.Channel_8.Input <-> Channel 8/Input
//     PlcTask Inputs/GVL_iXlinker.EtherCAT_Master_BKCUCX.TcTerminals210_EK1100_1.TcTerminals210_1BK1250.A_0180_KM_1002_16_Ch_Input_24V_3_0ms.Channel_9.Input <-> Channel 9/Input
//     PlcTask Inputs/GVL_iXlinker.EtherCAT_Master_BKCUCX.TcTerminals210_EK1100_1.TcTerminals210_1BK1250.A_0180_KM_1002_16_Ch_Input_24V_3_0ms.Channel_10.Input <-> Channel 10/Input
//     PlcTask Inputs/GVL_iXlinker.EtherCAT_Master_BKCUCX.TcTerminals210_EK1100_1.TcTerminals210_1BK1250.A_0180_KM_1002_16_Ch_Input_24V_3_0ms.Channel_11.Input <-> Channel 11/Input
//     PlcTask Inputs/GVL_iXlinker.EtherCAT_Master_BKCUCX.TcTerminals210_EK1100_1.TcTerminals210_1BK1250.A_0180_KM_1002_16_Ch_Input_24V_3_0ms.Channel_12.Input <-> Channel 12/Input
//     PlcTask Inputs/GVL_iXlinker.EtherCAT_Master_BKCUCX.TcTerminals210_EK1100_1.TcTerminals210_1BK1250.A_0180_KM_1002_16_Ch_Input_24V_3_0ms.Channel_13.Input <-> Channel 13/Input
//     PlcTask Inputs/GVL_iXlinker.EtherCAT_Master_BKCUCX.TcTerminals210_EK1100_1.TcTerminals210_1BK1250.A_0180_KM_1002_16_Ch_Input_24V_3_0ms.Channel_14.Input <-> Channel 14/Input
//     PlcTask Inputs/GVL_iXlinker.EtherCAT_Master_BKCUCX.TcTerminals210_EK1100_1.TcTerminals210_1BK1250.A_0180_KM_1002_16_Ch_Input_24V_3_0ms.Channel_15.Input <-> Channel 15/Input
//     PlcTask Inputs/GVL_iXlinker.EtherCAT_Master_BKCUCX.TcTerminals210_EK1100_1.TcTerminals210_1BK1250.A_0180_KM_1002_16_Ch_Input_24V_3_0ms.Channel_16.Input <-> Channel 16/Input
//   PLC/PLC Instance <-> EtherCAT Master BKCUCX/TcTerminals210_EK1100_1/TcTerminals210_1BK1250/A_0181(KM 1004, 32 Ch. Input (24V, 3.0ms))
//     PlcTask Inputs/GVL_iXlinker.EtherCAT_Master_BKCUCX.TcTerminals210_EK1100_1.TcTerminals210_1BK1250.A_0181_KM_1004_32_Ch_Input_24V_3_0ms.Channel_1.Input <-> Channel 1/Input
//     PlcTask Inputs/GVL_iXlinker.EtherCAT_Master_BKCUCX.TcTerminals210_EK1100_1.TcTerminals210_1BK1250.A_0181_KM_1004_32_Ch_Input_24V_3_0ms.Channel_2.Input <-> Channel 2/Input
//     PlcTask Inputs/GVL_iXlinker.EtherCAT_Master_BKCUCX.TcTerminals210_EK1100_1.TcTerminals210_1BK1250.A_0181_KM_1004_32_Ch_Input_24V_3_0ms.Channel_3.Input <-> Channel 3/Input
//     PlcTask Inputs/GVL_iXlinker.EtherCAT_Master_BKCUCX.TcTerminals210_EK1100_1.TcTerminals210_1BK1250.A_0181_KM_1004_32_Ch_Input_24V_3_0ms.Channel_4.Input <-> Channel 4/Input
//     PlcTask Inputs/GVL_iXlinker.EtherCAT_Master_BKCUCX.TcTerminals210_EK1100_1.TcTerminals210_1BK1250.A_0181_KM_1004_32_Ch_Input_24V_3_0ms.Channel_5.Input <-> Channel 5/Input
//     PlcTask Inputs/GVL_iXlinker.EtherCAT_Master_BKCUCX.TcTerminals210_EK1100_1.TcTerminals210_1BK1250.A_0181_KM_1004_32_Ch_Input_24V_3_0ms.Channel_6.Input <-> Channel 6/Input
//     PlcTask Inputs/GVL_iXlinker.EtherCAT_Master_BKCUCX.TcTerminals210_EK1100_1.TcTerminals210_1BK1250.A_0181_KM_1004_32_Ch_Input_24V_3_0ms.Channel_7.Input <-> Channel 7/Input
//     PlcTask Inputs/GVL_iXlinker.EtherCAT_Master_BKCUCX.TcTerminals210_EK1100_1.TcTerminals210_1BK1250.A_0181_KM_1004_32_Ch_Input_24V_3_0ms.Channel_8.Input <-> Channel 8/Input
//     PlcTask Inputs/GVL_iXlinker.EtherCAT_Master_BKCUCX.TcTerminals210_EK1100_1.TcTerminals210_1BK1250.A_0181_KM_1004_32_Ch_Input_24V_3_0ms.Channel_9.Input <-> Channel 9/Input
//     PlcTask Inputs/GVL_iXlinker.EtherCAT_Master_BKCUCX.TcTerminals210_EK1100_1.TcTerminals210_1BK1250.A_0181_KM_1004_32_Ch_Input_24V_3_0ms.Channel_10.Input <-> Channel 10/Input
//     PlcTask Inputs/GVL_iXlinker.EtherCAT_Master_BKCUCX.TcTerminals210_EK1100_1.TcTerminals210_1BK1250.A_0181_KM_1004_32_Ch_Input_24V_3_0ms.Channel_11.Input <-> Channel 11/Input
//     PlcTask Inputs/GVL_iXlinker.EtherCAT_Master_BKCUCX.TcTerminals210_EK1100_1.TcTerminals210_1BK1250.A_0181_KM_1004_32_Ch_Input_24V_3_0ms.Channel_12.Input <-> Channel 12/Input
//     PlcTask Inputs/GVL_iXlinker.EtherCAT_Master_BKCUCX.TcTerminals210_EK1100_1.TcTerminals210_1BK1250.A_0181_KM_1004_32_Ch_Input_24V_3_0ms.Channel_13.Input <-> Channel 13/Input
//     PlcTask Inputs/GVL_iXlinker.EtherCAT_Master_BKCUCX.TcTerminals210_EK1100_1.TcTerminals210_1BK1250.A_0181_KM_1004_32_Ch_Input_24V_3_0ms.Channel_14.Input <-> Channel 14/Input
//     PlcTask Inputs/GVL_iXlinker.EtherCAT_Master_BKCUCX.TcTerminals210_EK1100_1.TcTerminals210_1BK1250.A_0181_KM_1004_32_Ch_Input_24V_3_0ms.Channel_15.Input <-> Channel 15/Input
//     PlcTask Inputs/GVL_iXlinker.EtherCAT_Master_BKCUCX.TcTerminals210_EK1100_1.TcTerminals210_1BK1250.A_0181_KM_1004_32_Ch_Input_24V_3_0ms.Channel_16.Input <-> Channel 16/Input
//     PlcTask Inputs/GVL_iXlinker.EtherCAT_Master_BKCUCX.TcTerminals210_EK1100_1.TcTerminals210_1BK1250.A_0181_KM_1004_32_Ch_Input_24V_3_0ms.Channel_17.Input <-> Channel 17/Input
//     PlcTask Inputs/GVL_iXlinker.EtherCAT_Master_BKCUCX.TcTerminals210_EK1100_1.TcTerminals210_1BK1250.A_0181_KM_1004_32_Ch_Input_24V_3_0ms.Channel_18.Input <-> Channel 18/Input
//     PlcTask Inputs/GVL_iXlinker.EtherCAT_Master_BKCUCX.TcTerminals210_EK1100_1.TcTerminals210_1BK1250.A_0181_KM_1004_32_Ch_Input_24V_3_0ms.Channel_19.Input <-> Channel 19/Input
//     PlcTask Inputs/GVL_iXlinker.EtherCAT_Master_BKCUCX.TcTerminals210_EK1100_1.TcTerminals210_1BK1250.A_0181_KM_1004_32_Ch_Input_24V_3_0ms.Channel_20.Input <-> Channel 20/Input
//     PlcTask Inputs/GVL_iXlinker.EtherCAT_Master_BKCUCX.TcTerminals210_EK1100_1.TcTerminals210_1BK1250.A_0181_KM_1004_32_Ch_Input_24V_3_0ms.Channel_21.Input <-> Channel 21/Input
//     PlcTask Inputs/GVL_iXlinker.EtherCAT_Master_BKCUCX.TcTerminals210_EK1100_1.TcTerminals210_1BK1250.A_0181_KM_1004_32_Ch_Input_24V_3_0ms.Channel_22.Input <-> Channel 22/Input
//     PlcTask Inputs/GVL_iXlinker.EtherCAT_Master_BKCUCX.TcTerminals210_EK1100_1.TcTerminals210_1BK1250.A_0181_KM_1004_32_Ch_Input_24V_3_0ms.Channel_23.Input <-> Channel 23/Input
//     PlcTask Inputs/GVL_iXlinker.EtherCAT_Master_BKCUCX.TcTerminals210_EK1100_1.TcTerminals210_1BK1250.A_0181_KM_1004_32_Ch_Input_24V_3_0ms.Channel_24.Input <-> Channel 24/Input
//     PlcTask Inputs/GVL_iXlinker.EtherCAT_Master_BKCUCX.TcTerminals210_EK1100_1.TcTerminals210_1BK1250.A_0181_KM_1004_32_Ch_Input_24V_3_0ms.Channel_25.Input <-> Channel 25/Input
//     PlcTask Inputs/GVL_iXlinker.EtherCAT_Master_BKCUCX.TcTerminals210_EK1100_1.TcTerminals210_1BK1250.A_0181_KM_1004_32_Ch_Input_24V_3_0ms.Channel_26.Input <-> Channel 26/Input
//     PlcTask Inputs/GVL_iXlinker.EtherCAT_Master_BKCUCX.TcTerminals210_EK1100_1.TcTerminals210_1BK1250.A_0181_KM_1004_32_Ch_Input_24V_3_0ms.Channel_27.Input <-> Channel 27/Input
//     PlcTask Inputs/GVL_iXlinker.EtherCAT_Master_BKCUCX.TcTerminals210_EK1100_1.TcTerminals210_1BK1250.A_0181_KM_1004_32_Ch_Input_24V_3_0ms.Channel_28.Input <-> Channel 28/Input
//     PlcTask Inputs/GVL_iXlinker.EtherCAT_Master_BKCUCX.TcTerminals210_EK1100_1.TcTerminals210_1BK1250.A_0181_KM_1004_32_Ch_Input_24V_3_0ms.Channel_29.Input <-> Channel 29/Input
//     PlcTask Inputs/GVL_iXlinker.EtherCAT_Master_BKCUCX.TcTerminals210_EK1100_1.TcTerminals210_1BK1250.A_0181_KM_1004_32_Ch_Input_24V_3_0ms.Channel_30.Input <-> Channel 30/Input
//     PlcTask Inputs/GVL_iXlinker.EtherCAT_Master_BKCUCX.TcTerminals210_EK1100_1.TcTerminals210_1BK1250.A_0181_KM_1004_32_Ch_Input_24V_3_0ms.Channel_31.Input <-> Channel 31/Input
//     PlcTask Inputs/GVL_iXlinker.EtherCAT_Master_BKCUCX.TcTerminals210_EK1100_1.TcTerminals210_1BK1250.A_0181_KM_1004_32_Ch_Input_24V_3_0ms.Channel_32.Input <-> Channel 32/Input
//   PLC/PLC Instance <-> EtherCAT Master BKCUCX/TcTerminals210_EK1100_1/TcTerminals210_1BK1250/A_0182(KM 1008, 64 Ch. Input (24V, 3.0ms))
//     PlcTask Inputs/GVL_iXlinker.EtherCAT_Master_BKCUCX.TcTerminals210_EK1100_1.TcTerminals210_1BK1250.A_0182_KM_1008_64_Ch_Input_24V_3_0ms.Channel_1.Input <-> Channel 1/Input
//     PlcTask Inputs/GVL_iXlinker.EtherCAT_Master_BKCUCX.TcTerminals210_EK1100_1.TcTerminals210_1BK1250.A_0182_KM_1008_64_Ch_Input_24V_3_0ms.Channel_2.Input <-> Channel 2/Input
//     PlcTask Inputs/GVL_iXlinker.EtherCAT_Master_BKCUCX.TcTerminals210_EK1100_1.TcTerminals210_1BK1250.A_0182_KM_1008_64_Ch_Input_24V_3_0ms.Channel_3.Input <-> Channel 3/Input
//     PlcTask Inputs/GVL_iXlinker.EtherCAT_Master_BKCUCX.TcTerminals210_EK1100_1.TcTerminals210_1BK1250.A_0182_KM_1008_64_Ch_Input_24V_3_0ms.Channel_4.Input <-> Channel 4/Input
//     PlcTask Inputs/GVL_iXlinker.EtherCAT_Master_BKCUCX.TcTerminals210_EK1100_1.TcTerminals210_1BK1250.A_0182_KM_1008_64_Ch_Input_24V_3_0ms.Channel_5.Input <-> Channel 5/Input
//     PlcTask Inputs/GVL_iXlinker.EtherCAT_Master_BKCUCX.TcTerminals210_EK1100_1.TcTerminals210_1BK1250.A_0182_KM_1008_64_Ch_Input_24V_3_0ms.Channel_6.Input <-> Channel 6/Input
//     PlcTask Inputs/GVL_iXlinker.EtherCAT_Master_BKCUCX.TcTerminals210_EK1100_1.TcTerminals210_1BK1250.A_0182_KM_1008_64_Ch_Input_24V_3_0ms.Channel_7.Input <-> Channel 7/Input
//     PlcTask Inputs/GVL_iXlinker.EtherCAT_Master_BKCUCX.TcTerminals210_EK1100_1.TcTerminals210_1BK1250.A_0182_KM_1008_64_Ch_Input_24V_3_0ms.Channel_8.Input <-> Channel 8/Input
//     PlcTask Inputs/GVL_iXlinker.EtherCAT_Master_BKCUCX.TcTerminals210_EK1100_1.TcTerminals210_1BK1250.A_0182_KM_1008_64_Ch_Input_24V_3_0ms.Channel_9.Input <-> Channel 9/Input
//     PlcTask Inputs/GVL_iXlinker.EtherCAT_Master_BKCUCX.TcTerminals210_EK1100_1.TcTerminals210_1BK1250.A_0182_KM_1008_64_Ch_Input_24V_3_0ms.Channel_10.Input <-> Channel 10/Input
//     PlcTask Inputs/GVL_iXlinker.EtherCAT_Master_BKCUCX.TcTerminals210_EK1100_1.TcTerminals210_1BK1250.A_0182_KM_1008_64_Ch_Input_24V_3_0ms.Channel_11.Input <-> Channel 11/Input
//     PlcTask Inputs/GVL_iXlinker.EtherCAT_Master_BKCUCX.TcTerminals210_EK1100_1.TcTerminals210_1BK1250.A_0182_KM_1008_64_Ch_Input_24V_3_0ms.Channel_12.Input <-> Channel 12/Input
//     PlcTask Inputs/GVL_iXlinker.EtherCAT_Master_BKCUCX.TcTerminals210_EK1100_1.TcTerminals210_1BK1250.A_0182_KM_1008_64_Ch_Input_24V_3_0ms.Channel_13.Input <-> Channel 13/Input
//     PlcTask Inputs/GVL_iXlinker.EtherCAT_Master_BKCUCX.TcTerminals210_EK1100_1.TcTerminals210_1BK1250.A_0182_KM_1008_64_Ch_Input_24V_3_0ms.Channel_14.Input <-> Channel 14/Input
//     PlcTask Inputs/GVL_iXlinker.EtherCAT_Master_BKCUCX.TcTerminals210_EK1100_1.TcTerminals210_1BK1250.A_0182_KM_1008_64_Ch_Input_24V_3_0ms.Channel_15.Input <-> Channel 15/Input
//     PlcTask Inputs/GVL_iXlinker.EtherCAT_Master_BKCUCX.TcTerminals210_EK1100_1.TcTerminals210_1BK1250.A_0182_KM_1008_64_Ch_Input_24V_3_0ms.Channel_16.Input <-> Channel 16/Input
//     PlcTask Inputs/GVL_iXlinker.EtherCAT_Master_BKCUCX.TcTerminals210_EK1100_1.TcTerminals210_1BK1250.A_0182_KM_1008_64_Ch_Input_24V_3_0ms.Channel_17.Input <-> Channel 17/Input
//     PlcTask Inputs/GVL_iXlinker.EtherCAT_Master_BKCUCX.TcTerminals210_EK1100_1.TcTerminals210_1BK1250.A_0182_KM_1008_64_Ch_Input_24V_3_0ms.Channel_18.Input <-> Channel 18/Input
//     PlcTask Inputs/GVL_iXlinker.EtherCAT_Master_BKCUCX.TcTerminals210_EK1100_1.TcTerminals210_1BK1250.A_0182_KM_1008_64_Ch_Input_24V_3_0ms.Channel_19.Input <-> Channel 19/Input
//     PlcTask Inputs/GVL_iXlinker.EtherCAT_Master_BKCUCX.TcTerminals210_EK1100_1.TcTerminals210_1BK1250.A_0182_KM_1008_64_Ch_Input_24V_3_0ms.Channel_20.Input <-> Channel 20/Input
//     PlcTask Inputs/GVL_iXlinker.EtherCAT_Master_BKCUCX.TcTerminals210_EK1100_1.TcTerminals210_1BK1250.A_0182_KM_1008_64_Ch_Input_24V_3_0ms.Channel_21.Input <-> Channel 21/Input
//     PlcTask Inputs/GVL_iXlinker.EtherCAT_Master_BKCUCX.TcTerminals210_EK1100_1.TcTerminals210_1BK1250.A_0182_KM_1008_64_Ch_Input_24V_3_0ms.Channel_22.Input <-> Channel 22/Input
//     PlcTask Inputs/GVL_iXlinker.EtherCAT_Master_BKCUCX.TcTerminals210_EK1100_1.TcTerminals210_1BK1250.A_0182_KM_1008_64_Ch_Input_24V_3_0ms.Channel_23.Input <-> Channel 23/Input
//     PlcTask Inputs/GVL_iXlinker.EtherCAT_Master_BKCUCX.TcTerminals210_EK1100_1.TcTerminals210_1BK1250.A_0182_KM_1008_64_Ch_Input_24V_3_0ms.Channel_24.Input <-> Channel 24/Input
//     PlcTask Inputs/GVL_iXlinker.EtherCAT_Master_BKCUCX.TcTerminals210_EK1100_1.TcTerminals210_1BK1250.A_0182_KM_1008_64_Ch_Input_24V_3_0ms.Channel_25.Input <-> Channel 25/Input
//     PlcTask Inputs/GVL_iXlinker.EtherCAT_Master_BKCUCX.TcTerminals210_EK1100_1.TcTerminals210_1BK1250.A_0182_KM_1008_64_Ch_Input_24V_3_0ms.Channel_26.Input <-> Channel 26/Input
//     PlcTask Inputs/GVL_iXlinker.EtherCAT_Master_BKCUCX.TcTerminals210_EK1100_1.TcTerminals210_1BK1250.A_0182_KM_1008_64_Ch_Input_24V_3_0ms.Channel_27.Input <-> Channel 27/Input
//     PlcTask Inputs/GVL_iXlinker.EtherCAT_Master_BKCUCX.TcTerminals210_EK1100_1.TcTerminals210_1BK1250.A_0182_KM_1008_64_Ch_Input_24V_3_0ms.Channel_28.Input <-> Channel 28/Input
//     PlcTask Inputs/GVL_iXlinker.EtherCAT_Master_BKCUCX.TcTerminals210_EK1100_1.TcTerminals210_1BK1250.A_0182_KM_1008_64_Ch_Input_24V_3_0ms.Channel_29.Input <-> Channel 29/Input
//     PlcTask Inputs/GVL_iXlinker.EtherCAT_Master_BKCUCX.TcTerminals210_EK1100_1.TcTerminals210_1BK1250.A_0182_KM_1008_64_Ch_Input_24V_3_0ms.Channel_30.Input <-> Channel 30/Input
//     PlcTask Inputs/GVL_iXlinker.EtherCAT_Master_BKCUCX.TcTerminals210_EK1100_1.TcTerminals210_1BK1250.A_0182_KM_1008_64_Ch_Input_24V_3_0ms.Channel_31.Input <-> Channel 31/Input
//     PlcTask Inputs/GVL_iXlinker.EtherCAT_Master_BKCUCX.TcTerminals210_EK1100_1.TcTerminals210_1BK1250.A_0182_KM_1008_64_Ch_Input_24V_3_0ms.Channel_32.Input <-> Channel 32/Input
//     PlcTask Inputs/GVL_iXlinker.EtherCAT_Master_BKCUCX.TcTerminals210_EK1100_1.TcTerminals210_1BK1250.A_0182_KM_1008_64_Ch_Input_24V_3_0ms.Channel_33.Input <-> Channel 33/Input
//     PlcTask Inputs/GVL_iXlinker.EtherCAT_Master_BKCUCX.TcTerminals210_EK1100_1.TcTerminals210_1BK1250.A_0182_KM_1008_64_Ch_Input_24V_3_0ms.Channel_34.Input <-> Channel 34/Input
//     PlcTask Inputs/GVL_iXlinker.EtherCAT_Master_BKCUCX.TcTerminals210_EK1100_1.TcTerminals210_1BK1250.A_0182_KM_1008_64_Ch_Input_24V_3_0ms.Channel_35.Input <-> Channel 35/Input
//     PlcTask Inputs/GVL_iXlinker.EtherCAT_Master_BKCUCX.TcTerminals210_EK1100_1.TcTerminals210_1BK1250.A_0182_KM_1008_64_Ch_Input_24V_3_0ms.Channel_36.Input <-> Channel 36/Input
//     PlcTask Inputs/GVL_iXlinker.EtherCAT_Master_BKCUCX.TcTerminals210_EK1100_1.TcTerminals210_1BK1250.A_0182_KM_1008_64_Ch_Input_24V_3_0ms.Channel_37.Input <-> Channel 37/Input
//     PlcTask Inputs/GVL_iXlinker.EtherCAT_Master_BKCUCX.TcTerminals210_EK1100_1.TcTerminals210_1BK1250.A_0182_KM_1008_64_Ch_Input_24V_3_0ms.Channel_38.Input <-> Channel 38/Input
//     PlcTask Inputs/GVL_iXlinker.EtherCAT_Master_BKCUCX.TcTerminals210_EK1100_1.TcTerminals210_1BK1250.A_0182_KM_1008_64_Ch_Input_24V_3_0ms.Channel_39.Input <-> Channel 39/Input
//     PlcTask Inputs/GVL_iXlinker.EtherCAT_Master_BKCUCX.TcTerminals210_EK1100_1.TcTerminals210_1BK1250.A_0182_KM_1008_64_Ch_Input_24V_3_0ms.Channel_40.Input <-> Channel 40/Input
//     PlcTask Inputs/GVL_iXlinker.EtherCAT_Master_BKCUCX.TcTerminals210_EK1100_1.TcTerminals210_1BK1250.A_0182_KM_1008_64_Ch_Input_24V_3_0ms.Channel_41.Input <-> Channel 41/Input
//     PlcTask Inputs/GVL_iXlinker.EtherCAT_Master_BKCUCX.TcTerminals210_EK1100_1.TcTerminals210_1BK1250.A_0182_KM_1008_64_Ch_Input_24V_3_0ms.Channel_42.Input <-> Channel 42/Input
//     PlcTask Inputs/GVL_iXlinker.EtherCAT_Master_BKCUCX.TcTerminals210_EK1100_1.TcTerminals210_1BK1250.A_0182_KM_1008_64_Ch_Input_24V_3_0ms.Channel_43.Input <-> Channel 43/Input
//     PlcTask Inputs/GVL_iXlinker.EtherCAT_Master_BKCUCX.TcTerminals210_EK1100_1.TcTerminals210_1BK1250.A_0182_KM_1008_64_Ch_Input_24V_3_0ms.Channel_44.Input <-> Channel 44/Input
//     PlcTask Inputs/GVL_iXlinker.EtherCAT_Master_BKCUCX.TcTerminals210_EK1100_1.TcTerminals210_1BK1250.A_0182_KM_1008_64_Ch_Input_24V_3_0ms.Channel_45.Input <-> Channel 45/Input
//     PlcTask Inputs/GVL_iXlinker.EtherCAT_Master_BKCUCX.TcTerminals210_EK1100_1.TcTerminals210_1BK1250.A_0182_KM_1008_64_Ch_Input_24V_3_0ms.Channel_46.Input <-> Channel 46/Input
//     PlcTask Inputs/GVL_iXlinker.EtherCAT_Master_BKCUCX.TcTerminals210_EK1100_1.TcTerminals210_1BK1250.A_0182_KM_1008_64_Ch_Input_24V_3_0ms.Channel_47.Input <-> Channel 47/Input
//     PlcTask Inputs/GVL_iXlinker.EtherCAT_Master_BKCUCX.TcTerminals210_EK1100_1.TcTerminals210_1BK1250.A_0182_KM_1008_64_Ch_Input_24V_3_0ms.Channel_48.Input <-> Channel 48/Input
//     PlcTask Inputs/GVL_iXlinker.EtherCAT_Master_BKCUCX.TcTerminals210_EK1100_1.TcTerminals210_1BK1250.A_0182_KM_1008_64_Ch_Input_24V_3_0ms.Channel_49.Input <-> Channel 49/Input
//     PlcTask Inputs/GVL_iXlinker.EtherCAT_Master_BKCUCX.TcTerminals210_EK1100_1.TcTerminals210_1BK1250.A_0182_KM_1008_64_Ch_Input_24V_3_0ms.Channel_50.Input <-> Channel 50/Input
//     PlcTask Inputs/GVL_iXlinker.EtherCAT_Master_BKCUCX.TcTerminals210_EK1100_1.TcTerminals210_1BK1250.A_0182_KM_1008_64_Ch_Input_24V_3_0ms.Channel_51.Input <-> Channel 51/Input
//     PlcTask Inputs/GVL_iXlinker.EtherCAT_Master_BKCUCX.TcTerminals210_EK1100_1.TcTerminals210_1BK1250.A_0182_KM_1008_64_Ch_Input_24V_3_0ms.Channel_52.Input <-> Channel 52/Input
//     PlcTask Inputs/GVL_iXlinker.EtherCAT_Master_BKCUCX.TcTerminals210_EK1100_1.TcTerminals210_1BK1250.A_0182_KM_1008_64_Ch_Input_24V_3_0ms.Channel_53.Input <-> Channel 53/Input
//     PlcTask Inputs/GVL_iXlinker.EtherCAT_Master_BKCUCX.TcTerminals210_EK1100_1.TcTerminals210_1BK1250.A_0182_KM_1008_64_Ch_Input_24V_3_0ms.Channel_54.Input <-> Channel 54/Input
//     PlcTask Inputs/GVL_iXlinker.EtherCAT_Master_BKCUCX.TcTerminals210_EK1100_1.TcTerminals210_1BK1250.A_0182_KM_1008_64_Ch_Input_24V_3_0ms.Channel_55.Input <-> Channel 55/Input
//     PlcTask Inputs/GVL_iXlinker.EtherCAT_Master_BKCUCX.TcTerminals210_EK1100_1.TcTerminals210_1BK1250.A_0182_KM_1008_64_Ch_Input_24V_3_0ms.Channel_56.Input <-> Channel 56/Input
//     PlcTask Inputs/GVL_iXlinker.EtherCAT_Master_BKCUCX.TcTerminals210_EK1100_1.TcTerminals210_1BK1250.A_0182_KM_1008_64_Ch_Input_24V_3_0ms.Channel_57.Input <-> Channel 57/Input
//     PlcTask Inputs/GVL_iXlinker.EtherCAT_Master_BKCUCX.TcTerminals210_EK1100_1.TcTerminals210_1BK1250.A_0182_KM_1008_64_Ch_Input_24V_3_0ms.Channel_58.Input <-> Channel 58/Input
//     PlcTask Inputs/GVL_iXlinker.EtherCAT_Master_BKCUCX.TcTerminals210_EK1100_1.TcTerminals210_1BK1250.A_0182_KM_1008_64_Ch_Input_24V_3_0ms.Channel_59.Input <-> Channel 59/Input
//     PlcTask Inputs/GVL_iXlinker.EtherCAT_Master_BKCUCX.TcTerminals210_EK1100_1.TcTerminals210_1BK1250.A_0182_KM_1008_64_Ch_Input_24V_3_0ms.Channel_60.Input <-> Channel 60/Input
//     PlcTask Inputs/GVL_iXlinker.EtherCAT_Master_BKCUCX.TcTerminals210_EK1100_1.TcTerminals210_1BK1250.A_0182_KM_1008_64_Ch_Input_24V_3_0ms.Channel_61.Input <-> Channel 61/Input
//     PlcTask Inputs/GVL_iXlinker.EtherCAT_Master_BKCUCX.TcTerminals210_EK1100_1.TcTerminals210_1BK1250.A_0182_KM_1008_64_Ch_Input_24V_3_0ms.Channel_62.Input <-> Channel 62/Input
//     PlcTask Inputs/GVL_iXlinker.EtherCAT_Master_BKCUCX.TcTerminals210_EK1100_1.TcTerminals210_1BK1250.A_0182_KM_1008_64_Ch_Input_24V_3_0ms.Channel_63.Input <-> Channel 63/Input
//     PlcTask Inputs/GVL_iXlinker.EtherCAT_Master_BKCUCX.TcTerminals210_EK1100_1.TcTerminals210_1BK1250.A_0182_KM_1008_64_Ch_Input_24V_3_0ms.Channel_64.Input <-> Channel 64/Input
//   PLC/PLC Instance <-> EtherCAT Master BKCUCX/TcTerminals210_EK1100_1/TcTerminals210_1BK1250/A_0183(KM 1012, 16 Ch. Input (24V, 0.2ms))
//     PlcTask Inputs/GVL_iXlinker.EtherCAT_Master_BKCUCX.TcTerminals210_EK1100_1.TcTerminals210_1BK1250.A_0183_KM_1012_16_Ch_Input_24V_0_2ms.Channel_1.Input <-> Channel 1/Input
//     PlcTask Inputs/GVL_iXlinker.EtherCAT_Master_BKCUCX.TcTerminals210_EK1100_1.TcTerminals210_1BK1250.A_0183_KM_1012_16_Ch_Input_24V_0_2ms.Channel_2.Input <-> Channel 2/Input
//     PlcTask Inputs/GVL_iXlinker.EtherCAT_Master_BKCUCX.TcTerminals210_EK1100_1.TcTerminals210_1BK1250.A_0183_KM_1012_16_Ch_Input_24V_0_2ms.Channel_3.Input <-> Channel 3/Input
//     PlcTask Inputs/GVL_iXlinker.EtherCAT_Master_BKCUCX.TcTerminals210_EK1100_1.TcTerminals210_1BK1250.A_0183_KM_1012_16_Ch_Input_24V_0_2ms.Channel_4.Input <-> Channel 4/Input
//     PlcTask Inputs/GVL_iXlinker.EtherCAT_Master_BKCUCX.TcTerminals210_EK1100_1.TcTerminals210_1BK1250.A_0183_KM_1012_16_Ch_Input_24V_0_2ms.Channel_5.Input <-> Channel 5/Input
//     PlcTask Inputs/GVL_iXlinker.EtherCAT_Master_BKCUCX.TcTerminals210_EK1100_1.TcTerminals210_1BK1250.A_0183_KM_1012_16_Ch_Input_24V_0_2ms.Channel_6.Input <-> Channel 6/Input
//     PlcTask Inputs/GVL_iXlinker.EtherCAT_Master_BKCUCX.TcTerminals210_EK1100_1.TcTerminals210_1BK1250.A_0183_KM_1012_16_Ch_Input_24V_0_2ms.Channel_7.Input <-> Channel 7/Input
//     PlcTask Inputs/GVL_iXlinker.EtherCAT_Master_BKCUCX.TcTerminals210_EK1100_1.TcTerminals210_1BK1250.A_0183_KM_1012_16_Ch_Input_24V_0_2ms.Channel_8.Input <-> Channel 8/Input
//     PlcTask Inputs/GVL_iXlinker.EtherCAT_Master_BKCUCX.TcTerminals210_EK1100_1.TcTerminals210_1BK1250.A_0183_KM_1012_16_Ch_Input_24V_0_2ms.Channel_9.Input <-> Channel 9/Input
//     PlcTask Inputs/GVL_iXlinker.EtherCAT_Master_BKCUCX.TcTerminals210_EK1100_1.TcTerminals210_1BK1250.A_0183_KM_1012_16_Ch_Input_24V_0_2ms.Channel_10.Input <-> Channel 10/Input
//     PlcTask Inputs/GVL_iXlinker.EtherCAT_Master_BKCUCX.TcTerminals210_EK1100_1.TcTerminals210_1BK1250.A_0183_KM_1012_16_Ch_Input_24V_0_2ms.Channel_11.Input <-> Channel 11/Input
//     PlcTask Inputs/GVL_iXlinker.EtherCAT_Master_BKCUCX.TcTerminals210_EK1100_1.TcTerminals210_1BK1250.A_0183_KM_1012_16_Ch_Input_24V_0_2ms.Channel_12.Input <-> Channel 12/Input
//     PlcTask Inputs/GVL_iXlinker.EtherCAT_Master_BKCUCX.TcTerminals210_EK1100_1.TcTerminals210_1BK1250.A_0183_KM_1012_16_Ch_Input_24V_0_2ms.Channel_13.Input <-> Channel 13/Input
//     PlcTask Inputs/GVL_iXlinker.EtherCAT_Master_BKCUCX.TcTerminals210_EK1100_1.TcTerminals210_1BK1250.A_0183_KM_1012_16_Ch_Input_24V_0_2ms.Channel_14.Input <-> Channel 14/Input
//     PlcTask Inputs/GVL_iXlinker.EtherCAT_Master_BKCUCX.TcTerminals210_EK1100_1.TcTerminals210_1BK1250.A_0183_KM_1012_16_Ch_Input_24V_0_2ms.Channel_15.Input <-> Channel 15/Input
//     PlcTask Inputs/GVL_iXlinker.EtherCAT_Master_BKCUCX.TcTerminals210_EK1100_1.TcTerminals210_1BK1250.A_0183_KM_1012_16_Ch_Input_24V_0_2ms.Channel_16.Input <-> Channel 16/Input
//   PLC/PLC Instance <-> EtherCAT Master BKCUCX/TcTerminals210_EK1100_1/TcTerminals210_1BK1250/A_0184(KM 1014, 32 Ch. Input (24V, 0.2ms))
//     PlcTask Inputs/GVL_iXlinker.EtherCAT_Master_BKCUCX.TcTerminals210_EK1100_1.TcTerminals210_1BK1250.A_0184_KM_1014_32_Ch_Input_24V_0_2ms.Channel_1.Input <-> Channel 1/Input
//     PlcTask Inputs/GVL_iXlinker.EtherCAT_Master_BKCUCX.TcTerminals210_EK1100_1.TcTerminals210_1BK1250.A_0184_KM_1014_32_Ch_Input_24V_0_2ms.Channel_2.Input <-> Channel 2/Input
//     PlcTask Inputs/GVL_iXlinker.EtherCAT_Master_BKCUCX.TcTerminals210_EK1100_1.TcTerminals210_1BK1250.A_0184_KM_1014_32_Ch_Input_24V_0_2ms.Channel_3.Input <-> Channel 3/Input
//     PlcTask Inputs/GVL_iXlinker.EtherCAT_Master_BKCUCX.TcTerminals210_EK1100_1.TcTerminals210_1BK1250.A_0184_KM_1014_32_Ch_Input_24V_0_2ms.Channel_4.Input <-> Channel 4/Input
//     PlcTask Inputs/GVL_iXlinker.EtherCAT_Master_BKCUCX.TcTerminals210_EK1100_1.TcTerminals210_1BK1250.A_0184_KM_1014_32_Ch_Input_24V_0_2ms.Channel_5.Input <-> Channel 5/Input
//     PlcTask Inputs/GVL_iXlinker.EtherCAT_Master_BKCUCX.TcTerminals210_EK1100_1.TcTerminals210_1BK1250.A_0184_KM_1014_32_Ch_Input_24V_0_2ms.Channel_6.Input <-> Channel 6/Input
//     PlcTask Inputs/GVL_iXlinker.EtherCAT_Master_BKCUCX.TcTerminals210_EK1100_1.TcTerminals210_1BK1250.A_0184_KM_1014_32_Ch_Input_24V_0_2ms.Channel_7.Input <-> Channel 7/Input
//     PlcTask Inputs/GVL_iXlinker.EtherCAT_Master_BKCUCX.TcTerminals210_EK1100_1.TcTerminals210_1BK1250.A_0184_KM_1014_32_Ch_Input_24V_0_2ms.Channel_8.Input <-> Channel 8/Input
//     PlcTask Inputs/GVL_iXlinker.EtherCAT_Master_BKCUCX.TcTerminals210_EK1100_1.TcTerminals210_1BK1250.A_0184_KM_1014_32_Ch_Input_24V_0_2ms.Channel_9.Input <-> Channel 9/Input
//     PlcTask Inputs/GVL_iXlinker.EtherCAT_Master_BKCUCX.TcTerminals210_EK1100_1.TcTerminals210_1BK1250.A_0184_KM_1014_32_Ch_Input_24V_0_2ms.Channel_10.Input <-> Channel 10/Input
//     PlcTask Inputs/GVL_iXlinker.EtherCAT_Master_BKCUCX.TcTerminals210_EK1100_1.TcTerminals210_1BK1250.A_0184_KM_1014_32_Ch_Input_24V_0_2ms.Channel_11.Input <-> Channel 11/Input
//     PlcTask Inputs/GVL_iXlinker.EtherCAT_Master_BKCUCX.TcTerminals210_EK1100_1.TcTerminals210_1BK1250.A_0184_KM_1014_32_Ch_Input_24V_0_2ms.Channel_12.Input <-> Channel 12/Input
//     PlcTask Inputs/GVL_iXlinker.EtherCAT_Master_BKCUCX.TcTerminals210_EK1100_1.TcTerminals210_1BK1250.A_0184_KM_1014_32_Ch_Input_24V_0_2ms.Channel_13.Input <-> Channel 13/Input
//     PlcTask Inputs/GVL_iXlinker.EtherCAT_Master_BKCUCX.TcTerminals210_EK1100_1.TcTerminals210_1BK1250.A_0184_KM_1014_32_Ch_Input_24V_0_2ms.Channel_14.Input <-> Channel 14/Input
//     PlcTask Inputs/GVL_iXlinker.EtherCAT_Master_BKCUCX.TcTerminals210_EK1100_1.TcTerminals210_1BK1250.A_0184_KM_1014_32_Ch_Input_24V_0_2ms.Channel_15.Input <-> Channel 15/Input
//     PlcTask Inputs/GVL_iXlinker.EtherCAT_Master_BKCUCX.TcTerminals210_EK1100_1.TcTerminals210_1BK1250.A_0184_KM_1014_32_Ch_Input_24V_0_2ms.Channel_16.Input <-> Channel 16/Input
//     PlcTask Inputs/GVL_iXlinker.EtherCAT_Master_BKCUCX.TcTerminals210_EK1100_1.TcTerminals210_1BK1250.A_0184_KM_1014_32_Ch_Input_24V_0_2ms.Channel_17.Input <-> Channel 17/Input
//     PlcTask Inputs/GVL_iXlinker.EtherCAT_Master_BKCUCX.TcTerminals210_EK1100_1.TcTerminals210_1BK1250.A_0184_KM_1014_32_Ch_Input_24V_0_2ms.Channel_18.Input <-> Channel 18/Input
//     PlcTask Inputs/GVL_iXlinker.EtherCAT_Master_BKCUCX.TcTerminals210_EK1100_1.TcTerminals210_1BK1250.A_0184_KM_1014_32_Ch_Input_24V_0_2ms.Channel_19.Input <-> Channel 19/Input
//     PlcTask Inputs/GVL_iXlinker.EtherCAT_Master_BKCUCX.TcTerminals210_EK1100_1.TcTerminals210_1BK1250.A_0184_KM_1014_32_Ch_Input_24V_0_2ms.Channel_20.Input <-> Channel 20/Input
//     PlcTask Inputs/GVL_iXlinker.EtherCAT_Master_BKCUCX.TcTerminals210_EK1100_1.TcTerminals210_1BK1250.A_0184_KM_1014_32_Ch_Input_24V_0_2ms.Channel_21.Input <-> Channel 21/Input
//     PlcTask Inputs/GVL_iXlinker.EtherCAT_Master_BKCUCX.TcTerminals210_EK1100_1.TcTerminals210_1BK1250.A_0184_KM_1014_32_Ch_Input_24V_0_2ms.Channel_22.Input <-> Channel 22/Input
//     PlcTask Inputs/GVL_iXlinker.EtherCAT_Master_BKCUCX.TcTerminals210_EK1100_1.TcTerminals210_1BK1250.A_0184_KM_1014_32_Ch_Input_24V_0_2ms.Channel_23.Input <-> Channel 23/Input
//     PlcTask Inputs/GVL_iXlinker.EtherCAT_Master_BKCUCX.TcTerminals210_EK1100_1.TcTerminals210_1BK1250.A_0184_KM_1014_32_Ch_Input_24V_0_2ms.Channel_24.Input <-> Channel 24/Input
//     PlcTask Inputs/GVL_iXlinker.EtherCAT_Master_BKCUCX.TcTerminals210_EK1100_1.TcTerminals210_1BK1250.A_0184_KM_1014_32_Ch_Input_24V_0_2ms.Channel_25.Input <-> Channel 25/Input
//     PlcTask Inputs/GVL_iXlinker.EtherCAT_Master_BKCUCX.TcTerminals210_EK1100_1.TcTerminals210_1BK1250.A_0184_KM_1014_32_Ch_Input_24V_0_2ms.Channel_26.Input <-> Channel 26/Input
//     PlcTask Inputs/GVL_iXlinker.EtherCAT_Master_BKCUCX.TcTerminals210_EK1100_1.TcTerminals210_1BK1250.A_0184_KM_1014_32_Ch_Input_24V_0_2ms.Channel_27.Input <-> Channel 27/Input
//     PlcTask Inputs/GVL_iXlinker.EtherCAT_Master_BKCUCX.TcTerminals210_EK1100_1.TcTerminals210_1BK1250.A_0184_KM_1014_32_Ch_Input_24V_0_2ms.Channel_28.Input <-> Channel 28/Input
//     PlcTask Inputs/GVL_iXlinker.EtherCAT_Master_BKCUCX.TcTerminals210_EK1100_1.TcTerminals210_1BK1250.A_0184_KM_1014_32_Ch_Input_24V_0_2ms.Channel_29.Input <-> Channel 29/Input
//     PlcTask Inputs/GVL_iXlinker.EtherCAT_Master_BKCUCX.TcTerminals210_EK1100_1.TcTerminals210_1BK1250.A_0184_KM_1014_32_Ch_Input_24V_0_2ms.Channel_30.Input <-> Channel 30/Input
//     PlcTask Inputs/GVL_iXlinker.EtherCAT_Master_BKCUCX.TcTerminals210_EK1100_1.TcTerminals210_1BK1250.A_0184_KM_1014_32_Ch_Input_24V_0_2ms.Channel_31.Input <-> Channel 31/Input
//     PlcTask Inputs/GVL_iXlinker.EtherCAT_Master_BKCUCX.TcTerminals210_EK1100_1.TcTerminals210_1BK1250.A_0184_KM_1014_32_Ch_Input_24V_0_2ms.Channel_32.Input <-> Channel 32/Input
//   PLC/PLC Instance <-> EtherCAT Master BKCUCX/TcTerminals210_EK1100_1/TcTerminals210_1BK1250/A_0185(KM 1018, 64 Ch. Input (24V, 0.2ms))
//     PlcTask Inputs/GVL_iXlinker.EtherCAT_Master_BKCUCX.TcTerminals210_EK1100_1.TcTerminals210_1BK1250.A_0185_KM_1018_64_Ch_Input_24V_0_2ms.Channel_1.Input <-> Channel 1/Input
//     PlcTask Inputs/GVL_iXlinker.EtherCAT_Master_BKCUCX.TcTerminals210_EK1100_1.TcTerminals210_1BK1250.A_0185_KM_1018_64_Ch_Input_24V_0_2ms.Channel_2.Input <-> Channel 2/Input
//     PlcTask Inputs/GVL_iXlinker.EtherCAT_Master_BKCUCX.TcTerminals210_EK1100_1.TcTerminals210_1BK1250.A_0185_KM_1018_64_Ch_Input_24V_0_2ms.Channel_3.Input <-> Channel 3/Input
//     PlcTask Inputs/GVL_iXlinker.EtherCAT_Master_BKCUCX.TcTerminals210_EK1100_1.TcTerminals210_1BK1250.A_0185_KM_1018_64_Ch_Input_24V_0_2ms.Channel_4.Input <-> Channel 4/Input
//     PlcTask Inputs/GVL_iXlinker.EtherCAT_Master_BKCUCX.TcTerminals210_EK1100_1.TcTerminals210_1BK1250.A_0185_KM_1018_64_Ch_Input_24V_0_2ms.Channel_5.Input <-> Channel 5/Input
//     PlcTask Inputs/GVL_iXlinker.EtherCAT_Master_BKCUCX.TcTerminals210_EK1100_1.TcTerminals210_1BK1250.A_0185_KM_1018_64_Ch_Input_24V_0_2ms.Channel_6.Input <-> Channel 6/Input
//     PlcTask Inputs/GVL_iXlinker.EtherCAT_Master_BKCUCX.TcTerminals210_EK1100_1.TcTerminals210_1BK1250.A_0185_KM_1018_64_Ch_Input_24V_0_2ms.Channel_7.Input <-> Channel 7/Input
//     PlcTask Inputs/GVL_iXlinker.EtherCAT_Master_BKCUCX.TcTerminals210_EK1100_1.TcTerminals210_1BK1250.A_0185_KM_1018_64_Ch_Input_24V_0_2ms.Channel_8.Input <-> Channel 8/Input
//     PlcTask Inputs/GVL_iXlinker.EtherCAT_Master_BKCUCX.TcTerminals210_EK1100_1.TcTerminals210_1BK1250.A_0185_KM_1018_64_Ch_Input_24V_0_2ms.Channel_9.Input <-> Channel 9/Input
//     PlcTask Inputs/GVL_iXlinker.EtherCAT_Master_BKCUCX.TcTerminals210_EK1100_1.TcTerminals210_1BK1250.A_0185_KM_1018_64_Ch_Input_24V_0_2ms.Channel_10.Input <-> Channel 10/Input
//     PlcTask Inputs/GVL_iXlinker.EtherCAT_Master_BKCUCX.TcTerminals210_EK1100_1.TcTerminals210_1BK1250.A_0185_KM_1018_64_Ch_Input_24V_0_2ms.Channel_11.Input <-> Channel 11/Input
//     PlcTask Inputs/GVL_iXlinker.EtherCAT_Master_BKCUCX.TcTerminals210_EK1100_1.TcTerminals210_1BK1250.A_0185_KM_1018_64_Ch_Input_24V_0_2ms.Channel_12.Input <-> Channel 12/Input
//     PlcTask Inputs/GVL_iXlinker.EtherCAT_Master_BKCUCX.TcTerminals210_EK1100_1.TcTerminals210_1BK1250.A_0185_KM_1018_64_Ch_Input_24V_0_2ms.Channel_13.Input <-> Channel 13/Input
//     PlcTask Inputs/GVL_iXlinker.EtherCAT_Master_BKCUCX.TcTerminals210_EK1100_1.TcTerminals210_1BK1250.A_0185_KM_1018_64_Ch_Input_24V_0_2ms.Channel_14.Input <-> Channel 14/Input
//     PlcTask Inputs/GVL_iXlinker.EtherCAT_Master_BKCUCX.TcTerminals210_EK1100_1.TcTerminals210_1BK1250.A_0185_KM_1018_64_Ch_Input_24V_0_2ms.Channel_15.Input <-> Channel 15/Input
//     PlcTask Inputs/GVL_iXlinker.EtherCAT_Master_BKCUCX.TcTerminals210_EK1100_1.TcTerminals210_1BK1250.A_0185_KM_1018_64_Ch_Input_24V_0_2ms.Channel_16.Input <-> Channel 16/Input
//     PlcTask Inputs/GVL_iXlinker.EtherCAT_Master_BKCUCX.TcTerminals210_EK1100_1.TcTerminals210_1BK1250.A_0185_KM_1018_64_Ch_Input_24V_0_2ms.Channel_17.Input <-> Channel 17/Input
//     PlcTask Inputs/GVL_iXlinker.EtherCAT_Master_BKCUCX.TcTerminals210_EK1100_1.TcTerminals210_1BK1250.A_0185_KM_1018_64_Ch_Input_24V_0_2ms.Channel_18.Input <-> Channel 18/Input
//     PlcTask Inputs/GVL_iXlinker.EtherCAT_Master_BKCUCX.TcTerminals210_EK1100_1.TcTerminals210_1BK1250.A_0185_KM_1018_64_Ch_Input_24V_0_2ms.Channel_19.Input <-> Channel 19/Input
//     PlcTask Inputs/GVL_iXlinker.EtherCAT_Master_BKCUCX.TcTerminals210_EK1100_1.TcTerminals210_1BK1250.A_0185_KM_1018_64_Ch_Input_24V_0_2ms.Channel_20.Input <-> Channel 20/Input
//     PlcTask Inputs/GVL_iXlinker.EtherCAT_Master_BKCUCX.TcTerminals210_EK1100_1.TcTerminals210_1BK1250.A_0185_KM_1018_64_Ch_Input_24V_0_2ms.Channel_21.Input <-> Channel 21/Input
//     PlcTask Inputs/GVL_iXlinker.EtherCAT_Master_BKCUCX.TcTerminals210_EK1100_1.TcTerminals210_1BK1250.A_0185_KM_1018_64_Ch_Input_24V_0_2ms.Channel_22.Input <-> Channel 22/Input
//     PlcTask Inputs/GVL_iXlinker.EtherCAT_Master_BKCUCX.TcTerminals210_EK1100_1.TcTerminals210_1BK1250.A_0185_KM_1018_64_Ch_Input_24V_0_2ms.Channel_23.Input <-> Channel 23/Input
//     PlcTask Inputs/GVL_iXlinker.EtherCAT_Master_BKCUCX.TcTerminals210_EK1100_1.TcTerminals210_1BK1250.A_0185_KM_1018_64_Ch_Input_24V_0_2ms.Channel_24.Input <-> Channel 24/Input
//     PlcTask Inputs/GVL_iXlinker.EtherCAT_Master_BKCUCX.TcTerminals210_EK1100_1.TcTerminals210_1BK1250.A_0185_KM_1018_64_Ch_Input_24V_0_2ms.Channel_25.Input <-> Channel 25/Input
//     PlcTask Inputs/GVL_iXlinker.EtherCAT_Master_BKCUCX.TcTerminals210_EK1100_1.TcTerminals210_1BK1250.A_0185_KM_1018_64_Ch_Input_24V_0_2ms.Channel_26.Input <-> Channel 26/Input
//     PlcTask Inputs/GVL_iXlinker.EtherCAT_Master_BKCUCX.TcTerminals210_EK1100_1.TcTerminals210_1BK1250.A_0185_KM_1018_64_Ch_Input_24V_0_2ms.Channel_27.Input <-> Channel 27/Input
//     PlcTask Inputs/GVL_iXlinker.EtherCAT_Master_BKCUCX.TcTerminals210_EK1100_1.TcTerminals210_1BK1250.A_0185_KM_1018_64_Ch_Input_24V_0_2ms.Channel_28.Input <-> Channel 28/Input
//     PlcTask Inputs/GVL_iXlinker.EtherCAT_Master_BKCUCX.TcTerminals210_EK1100_1.TcTerminals210_1BK1250.A_0185_KM_1018_64_Ch_Input_24V_0_2ms.Channel_29.Input <-> Channel 29/Input
//     PlcTask Inputs/GVL_iXlinker.EtherCAT_Master_BKCUCX.TcTerminals210_EK1100_1.TcTerminals210_1BK1250.A_0185_KM_1018_64_Ch_Input_24V_0_2ms.Channel_30.Input <-> Channel 30/Input
//     PlcTask Inputs/GVL_iXlinker.EtherCAT_Master_BKCUCX.TcTerminals210_EK1100_1.TcTerminals210_1BK1250.A_0185_KM_1018_64_Ch_Input_24V_0_2ms.Channel_31.Input <-> Channel 31/Input
//     PlcTask Inputs/GVL_iXlinker.EtherCAT_Master_BKCUCX.TcTerminals210_EK1100_1.TcTerminals210_1BK1250.A_0185_KM_1018_64_Ch_Input_24V_0_2ms.Channel_32.Input <-> Channel 32/Input
//     PlcTask Inputs/GVL_iXlinker.EtherCAT_Master_BKCUCX.TcTerminals210_EK1100_1.TcTerminals210_1BK1250.A_0185_KM_1018_64_Ch_Input_24V_0_2ms.Channel_33.Input <-> Channel 33/Input
//     PlcTask Inputs/GVL_iXlinker.EtherCAT_Master_BKCUCX.TcTerminals210_EK1100_1.TcTerminals210_1BK1250.A_0185_KM_1018_64_Ch_Input_24V_0_2ms.Channel_34.Input <-> Channel 34/Input
//     PlcTask Inputs/GVL_iXlinker.EtherCAT_Master_BKCUCX.TcTerminals210_EK1100_1.TcTerminals210_1BK1250.A_0185_KM_1018_64_Ch_Input_24V_0_2ms.Channel_35.Input <-> Channel 35/Input
//     PlcTask Inputs/GVL_iXlinker.EtherCAT_Master_BKCUCX.TcTerminals210_EK1100_1.TcTerminals210_1BK1250.A_0185_KM_1018_64_Ch_Input_24V_0_2ms.Channel_36.Input <-> Channel 36/Input
//     PlcTask Inputs/GVL_iXlinker.EtherCAT_Master_BKCUCX.TcTerminals210_EK1100_1.TcTerminals210_1BK1250.A_0185_KM_1018_64_Ch_Input_24V_0_2ms.Channel_37.Input <-> Channel 37/Input
//     PlcTask Inputs/GVL_iXlinker.EtherCAT_Master_BKCUCX.TcTerminals210_EK1100_1.TcTerminals210_1BK1250.A_0185_KM_1018_64_Ch_Input_24V_0_2ms.Channel_38.Input <-> Channel 38/Input
//     PlcTask Inputs/GVL_iXlinker.EtherCAT_Master_BKCUCX.TcTerminals210_EK1100_1.TcTerminals210_1BK1250.A_0185_KM_1018_64_Ch_Input_24V_0_2ms.Channel_39.Input <-> Channel 39/Input
//     PlcTask Inputs/GVL_iXlinker.EtherCAT_Master_BKCUCX.TcTerminals210_EK1100_1.TcTerminals210_1BK1250.A_0185_KM_1018_64_Ch_Input_24V_0_2ms.Channel_40.Input <-> Channel 40/Input
//     PlcTask Inputs/GVL_iXlinker.EtherCAT_Master_BKCUCX.TcTerminals210_EK1100_1.TcTerminals210_1BK1250.A_0185_KM_1018_64_Ch_Input_24V_0_2ms.Channel_41.Input <-> Channel 41/Input
//     PlcTask Inputs/GVL_iXlinker.EtherCAT_Master_BKCUCX.TcTerminals210_EK1100_1.TcTerminals210_1BK1250.A_0185_KM_1018_64_Ch_Input_24V_0_2ms.Channel_42.Input <-> Channel 42/Input
//     PlcTask Inputs/GVL_iXlinker.EtherCAT_Master_BKCUCX.TcTerminals210_EK1100_1.TcTerminals210_1BK1250.A_0185_KM_1018_64_Ch_Input_24V_0_2ms.Channel_43.Input <-> Channel 43/Input
//     PlcTask Inputs/GVL_iXlinker.EtherCAT_Master_BKCUCX.TcTerminals210_EK1100_1.TcTerminals210_1BK1250.A_0185_KM_1018_64_Ch_Input_24V_0_2ms.Channel_44.Input <-> Channel 44/Input
//     PlcTask Inputs/GVL_iXlinker.EtherCAT_Master_BKCUCX.TcTerminals210_EK1100_1.TcTerminals210_1BK1250.A_0185_KM_1018_64_Ch_Input_24V_0_2ms.Channel_45.Input <-> Channel 45/Input
//     PlcTask Inputs/GVL_iXlinker.EtherCAT_Master_BKCUCX.TcTerminals210_EK1100_1.TcTerminals210_1BK1250.A_0185_KM_1018_64_Ch_Input_24V_0_2ms.Channel_46.Input <-> Channel 46/Input
//     PlcTask Inputs/GVL_iXlinker.EtherCAT_Master_BKCUCX.TcTerminals210_EK1100_1.TcTerminals210_1BK1250.A_0185_KM_1018_64_Ch_Input_24V_0_2ms.Channel_47.Input <-> Channel 47/Input
//     PlcTask Inputs/GVL_iXlinker.EtherCAT_Master_BKCUCX.TcTerminals210_EK1100_1.TcTerminals210_1BK1250.A_0185_KM_1018_64_Ch_Input_24V_0_2ms.Channel_48.Input <-> Channel 48/Input
//     PlcTask Inputs/GVL_iXlinker.EtherCAT_Master_BKCUCX.TcTerminals210_EK1100_1.TcTerminals210_1BK1250.A_0185_KM_1018_64_Ch_Input_24V_0_2ms.Channel_49.Input <-> Channel 49/Input
//     PlcTask Inputs/GVL_iXlinker.EtherCAT_Master_BKCUCX.TcTerminals210_EK1100_1.TcTerminals210_1BK1250.A_0185_KM_1018_64_Ch_Input_24V_0_2ms.Channel_50.Input <-> Channel 50/Input
//     PlcTask Inputs/GVL_iXlinker.EtherCAT_Master_BKCUCX.TcTerminals210_EK1100_1.TcTerminals210_1BK1250.A_0185_KM_1018_64_Ch_Input_24V_0_2ms.Channel_51.Input <-> Channel 51/Input
//     PlcTask Inputs/GVL_iXlinker.EtherCAT_Master_BKCUCX.TcTerminals210_EK1100_1.TcTerminals210_1BK1250.A_0185_KM_1018_64_Ch_Input_24V_0_2ms.Channel_52.Input <-> Channel 52/Input
//     PlcTask Inputs/GVL_iXlinker.EtherCAT_Master_BKCUCX.TcTerminals210_EK1100_1.TcTerminals210_1BK1250.A_0185_KM_1018_64_Ch_Input_24V_0_2ms.Channel_53.Input <-> Channel 53/Input
//     PlcTask Inputs/GVL_iXlinker.EtherCAT_Master_BKCUCX.TcTerminals210_EK1100_1.TcTerminals210_1BK1250.A_0185_KM_1018_64_Ch_Input_24V_0_2ms.Channel_54.Input <-> Channel 54/Input
//     PlcTask Inputs/GVL_iXlinker.EtherCAT_Master_BKCUCX.TcTerminals210_EK1100_1.TcTerminals210_1BK1250.A_0185_KM_1018_64_Ch_Input_24V_0_2ms.Channel_55.Input <-> Channel 55/Input
//     PlcTask Inputs/GVL_iXlinker.EtherCAT_Master_BKCUCX.TcTerminals210_EK1100_1.TcTerminals210_1BK1250.A_0185_KM_1018_64_Ch_Input_24V_0_2ms.Channel_56.Input <-> Channel 56/Input
//     PlcTask Inputs/GVL_iXlinker.EtherCAT_Master_BKCUCX.TcTerminals210_EK1100_1.TcTerminals210_1BK1250.A_0185_KM_1018_64_Ch_Input_24V_0_2ms.Channel_57.Input <-> Channel 57/Input
//     PlcTask Inputs/GVL_iXlinker.EtherCAT_Master_BKCUCX.TcTerminals210_EK1100_1.TcTerminals210_1BK1250.A_0185_KM_1018_64_Ch_Input_24V_0_2ms.Channel_58.Input <-> Channel 58/Input
//     PlcTask Inputs/GVL_iXlinker.EtherCAT_Master_BKCUCX.TcTerminals210_EK1100_1.TcTerminals210_1BK1250.A_0185_KM_1018_64_Ch_Input_24V_0_2ms.Channel_59.Input <-> Channel 59/Input
//     PlcTask Inputs/GVL_iXlinker.EtherCAT_Master_BKCUCX.TcTerminals210_EK1100_1.TcTerminals210_1BK1250.A_0185_KM_1018_64_Ch_Input_24V_0_2ms.Channel_60.Input <-> Channel 60/Input
//     PlcTask Inputs/GVL_iXlinker.EtherCAT_Master_BKCUCX.TcTerminals210_EK1100_1.TcTerminals210_1BK1250.A_0185_KM_1018_64_Ch_Input_24V_0_2ms.Channel_61.Input <-> Channel 61/Input
//     PlcTask Inputs/GVL_iXlinker.EtherCAT_Master_BKCUCX.TcTerminals210_EK1100_1.TcTerminals210_1BK1250.A_0185_KM_1018_64_Ch_Input_24V_0_2ms.Channel_62.Input <-> Channel 62/Input
//     PlcTask Inputs/GVL_iXlinker.EtherCAT_Master_BKCUCX.TcTerminals210_EK1100_1.TcTerminals210_1BK1250.A_0185_KM_1018_64_Ch_Input_24V_0_2ms.Channel_63.Input <-> Channel 63/Input
//     PlcTask Inputs/GVL_iXlinker.EtherCAT_Master_BKCUCX.TcTerminals210_EK1100_1.TcTerminals210_1BK1250.A_0185_KM_1018_64_Ch_Input_24V_0_2ms.Channel_64.Input <-> Channel 64/Input
//   PLC/PLC Instance <-> EtherCAT Master BKCUCX/TcTerminals210_EK1100_1/TcTerminals210_1BK1250/A_0186(KM 1644, 4 Ch. Input, manual operation)
//     PlcTask Inputs/GVL_iXlinker.EtherCAT_Master_BKCUCX.TcTerminals210_EK1100_1.TcTerminals210_1BK1250.A_0186_KM_1644_4_Ch_Input_manual_operation.Channel_1.Switch <-> Channel 1/Switch
//     PlcTask Inputs/GVL_iXlinker.EtherCAT_Master_BKCUCX.TcTerminals210_EK1100_1.TcTerminals210_1BK1250.A_0186_KM_1644_4_Ch_Input_manual_operation.Channel_2.Switch <-> Channel 2/Switch
//     PlcTask Inputs/GVL_iXlinker.EtherCAT_Master_BKCUCX.TcTerminals210_EK1100_1.TcTerminals210_1BK1250.A_0186_KM_1644_4_Ch_Input_manual_operation.Channel_3.Switch <-> Channel 3/Switch
//     PlcTask Inputs/GVL_iXlinker.EtherCAT_Master_BKCUCX.TcTerminals210_EK1100_1.TcTerminals210_1BK1250.A_0186_KM_1644_4_Ch_Input_manual_operation.Channel_4.Switch <-> Channel 4/Switch
//     PlcTask Outputs/GVL_iXlinker.EtherCAT_Master_BKCUCX.TcTerminals210_EK1100_1.TcTerminals210_1BK1250.A_0186_KM_1644_4_Ch_Input_manual_operation.Channel_1.Output <-> Channel 1/Output
//     PlcTask Outputs/GVL_iXlinker.EtherCAT_Master_BKCUCX.TcTerminals210_EK1100_1.TcTerminals210_1BK1250.A_0186_KM_1644_4_Ch_Input_manual_operation.Channel_2.Output <-> Channel 2/Output
//     PlcTask Outputs/GVL_iXlinker.EtherCAT_Master_BKCUCX.TcTerminals210_EK1100_1.TcTerminals210_1BK1250.A_0186_KM_1644_4_Ch_Input_manual_operation.Channel_3.Output <-> Channel 3/Output
//     PlcTask Outputs/GVL_iXlinker.EtherCAT_Master_BKCUCX.TcTerminals210_EK1100_1.TcTerminals210_1BK1250.A_0186_KM_1644_4_Ch_Input_manual_operation.Channel_4.Output <-> Channel 4/Output
